	{attribute 'TcIecLibraryType'}
	{attribute 'external_name' := 'F_VN_TransformIntoDisplayableImage_GUID_02E0E048_CC89_5F60_6F70_D9022D4465A5'}
	(* Transform an image into a displayable image. The source image will be released and zeroed while existing destination images will be released and overwritten with the function result. The source image must not be used anywhere else and the transformation is very fast. If you want to use ipSrcImage after this function call, use F_VN_CopyIntoDisplayableImage instead. *)
	FUNCTION F_VN_TransformIntoDisplayableImage : HRESULT
	VAR_INPUT
		ipSrcImage	:	REFERENCE TO ITcVnImage;	(* Source image *)
		ipDestImage	:	REFERENCE TO ITcVnDisplayableImage;	(* Returns the displayable image *)
		hrPrev	:	HRESULT;	(* HRESULT indicating the result of previous operations (If SUCCEEDED(hrPrev) equals false, no operation is executed.) *)
	END_VAR

END_FUNCTION

// Functions/Basic Image Operations/F_VN_CreateAssociatedImage

	{attribute 'TcIecLibraryType'}
	{attribute 'external_name' := 'F_VN_CreateAssociatedImage_GUID_40D3B2A0_2CE9_5E22_5A39_BDDFD776A88E'}
	(* Creates a new image that shares its data with the source image. E.g. useful to work on different (disjoint) ROIs in parallel. *)
	FUNCTION F_VN_CreateAssociatedImage : HRESULT
	VAR_INPUT
		ipSrcImage	:	ITcVnImage;	(* Source image *)
		ipDestImage	:	REFERENCE TO ITcVnImage;	(* Returns the created image (Non-zero interface pointers are reused.) *)
		hrPrev	:	HRESULT;	(* HRESULT indicating the result of previous operations (If SUCCEEDED(hrPrev) equals false, no operation is executed.) *)
	END_VAR

END_FUNCTION

// Functions/Basic Image Operations/F_VN_CreateEmptyImage

	{attribute 'TcIecLibraryType'}
	{attribute 'external_name' := 'F_VN_CreateEmptyImage_GUID_87DE2717_AD60_5E53_651E_5AB98332C7FD'}
	(* Creates an empty image without allocating any data buffer. The initial reference count is set to one if a new image interface is created and kept, otherwise. *)
	FUNCTION F_VN_CreateEmptyImage : HRESULT
	VAR_INPUT
		ipImage	:	REFERENCE TO ITcVnImage;	(* Returns the created image *)
		hrPrev	:	HRESULT;	(* HRESULT indicating the result of previous operations (If SUCCEEDED(hrPrev) equals false, no operation is executed.) *)
	END_VAR

END_FUNCTION

// Functions/Basic Image Operations/F_VN_CreateImage

	{attribute 'TcIecLibraryType'}
	{attribute 'external_name' := 'F_VN_CreateImage_GUID_8D7420DD_6F30_56B3_5361_D2A5604ACF86'}
	(* Creates an image and allocate an appropriate data buffer. The initial reference count is set to one if a new image interface is created and kept, otherwise. *)
	FUNCTION F_VN_CreateImage : HRESULT
	VAR_INPUT
		ipImage	:	REFERENCE TO ITcVnImage;	(* Returns the created image (Non-zero interface pointers are reused.) *)
		nWidth	:	UDINT;	(* Image width *)
		nHeight	:	UDINT;	(* Image height *)
		ePixelType	:	ETcVnElementType;	(* Pixel type *)
		nChannelNum	:	UDINT;	(* Number of channels (1 to 255) *)
		hrPrev	:	HRESULT;	(* HRESULT indicating the result of previous operations (If SUCCEEDED(hrPrev) equals false, no operation is executed.) *)
	END_VAR

END_FUNCTION

// Functions/Basic Image Operations/F_VN_CreateImageAndSetPixels

	{attribute 'TcIecLibraryType'}
	{attribute 'external_name' := 'F_VN_CreateImageAndSetPixels_GUID_A8920FF8_8F96_5FBC_52F3_92CD14F74A4F'}
	(* Creates an image, allocates an appropriate data buffer and sets all pixels to the specified value. The initial reference count is set to one if a new image interface is created and kept, otherwise. *)
	FUNCTION F_VN_CreateImageAndSetPixels : HRESULT
	VAR_INPUT
		ipImage	:	REFERENCE TO ITcVnImage;	(* Returns the created image (Non-zero interface pointers are reused.) *)
		nWidth	:	UDINT;	(* Image width *)
		nHeight	:	UDINT;	(* Image height *)
		ePixelType	:	ETcVnElementType;	(* Pixel type *)
		nChannelNum	:	UDINT;	(* Number of channels (1 to 4) *)
		aValue	:	REFERENCE TO TcVnVector4_LREAL;	(* Pixel value *)
		hrPrev	:	HRESULT;	(* HRESULT indicating the result of previous operations (If SUCCEEDED(hrPrev) equals false, no operation is executed.) *)
	END_VAR

END_FUNCTION

// Functions/Basic Image Operations/F_VN_CreateImageFromArray

	{attribute 'TcIecLibraryType'}
	{attribute 'external_name' := 'F_VN_CreateImageFromArray_GUID_61CDDD3E_1106_53D6_5356_1EDFAEADE3E0'}
	(* Creates an image and initialize it with the provided data. The initial reference count is set to one if a new image interface is created and kept, otherwise. *)
	FUNCTION F_VN_CreateImageFromArray : HRESULT
	VAR_INPUT
		pData	:	PVOID;	(* Pointer to the 1D data array. Make sure that the array contains at least nWidth * nHeight * nChannelNum elements and that the array element type matches ePixelType. *)
		ipImage	:	REFERENCE TO ITcVnImage;	(* Returns the created image (Non-zero interface pointers are reused.) *)
		nWidth	:	UDINT;	(* Image width *)
		nHeight	:	UDINT;	(* Image height *)
		ePixelType	:	ETcVnElementType;	(* Pixel type *)
		nChannelNum	:	UDINT;	(* Number of channels (1 to 255) *)
		hrPrev	:	HRESULT;	(* HRESULT indicating the result of previous operations (If SUCCEEDED(hrPrev) equals false, no operation is executed.) *)
	END_VAR

END_FUNCTION

// Functions/Basic Image Operations/F_VN_ExportImage

	{attribute 'TcIecLibraryType'}
	{attribute 'external_name' := 'F_VN_ExportImage_GUID_12937EAB_04EC_5AB4_58D9_551F14B67CB3'}
	(* Exports the image data into a given buffer (e.g. an array). F_VN_ExportImageSize should be called before to get the required buffer size. *)
	FUNCTION F_VN_ExportImage : HRESULT
	VAR_INPUT
		ipImage	:	ITcVnImage;	(* Image *)
		pBuffer	:	PVOID;	(* Pointer to a buffer to store the image data (Make sure to allocate enough memory! The required size in bytes can be determined using the function F_VN_ExportImageSize) *)
		nBufferSize	:	ULINT;	(* Size of the buffer memory in bytes *)
		hrPrev	:	HRESULT;	(* HRESULT indicating the result of previous operations (If SUCCEEDED(hrPrev) equals false, no operation is executed.) *)
	END_VAR

END_FUNCTION

// Functions/Basic Image Operations/F_VN_ExportImageSize

	{attribute 'TcIecLibraryType'}
	{attribute 'external_name' := 'F_VN_ExportImageSize_GUID_992C005D_F63B_55F7_7FBB_93717F8A23F0'}
	(* Get the required buffer size (in bytes) to store the image data. *)
	FUNCTION F_VN_ExportImageSize : HRESULT
	VAR_INPUT
		ipImage	:	ITcVnImage;	(* Image *)
		nBufferSize	:	REFERENCE TO ULINT;	(* Returns the required buffer size in bytes *)
		hrPrev	:	HRESULT;	(* HRESULT indicating the result of previous operations (If SUCCEEDED(hrPrev) equals false, no operation is executed.) *)
	END_VAR

END_FUNCTION

// Functions/Basic Image Operations/F_VN_ExportImageAsBmp

	{attribute 'TcIecLibraryType'}
	{attribute 'external_name' := 'F_VN_ExportImageAsBmp_GUID_4BCA8984_D078_540E_761E_EBF20019EFCB'}
	(* Exports the image as bitmap into a given buffer (e.g. an array). F_VN_ExportImageAsBmpSize should be called before to get the required buffer size. *)
	FUNCTION F_VN_ExportImageAsBmp : HRESULT
	VAR_INPUT
		ipImage	:	ITcVnImage;	(* Image *)
		pBuffer	:	PVOID;	(* Pointer to a buffer to store the bitmap image (Make sure to allocate enough memory! The required size in bytes can be determined using the function F_VN_ExportImageAsBmpSize) *)
		nBufferSize	:	ULINT;	(* Size of the buffer memory in bytes *)
		hrPrev	:	HRESULT;	(* HRESULT indicating the result of previous operations (If SUCCEEDED(hrPrev) equals false, no operation is executed.) *)
	END_VAR

END_FUNCTION

// Functions/Basic Image Operations/F_VN_ExportImageAsBmpSize

	{attribute 'TcIecLibraryType'}
	{attribute 'external_name' := 'F_VN_ExportImageAsBmpSize_GUID_0FD9F0BD_DE92_5963_6C27_50E4417ED287'}
	(* Get the required buffer size (in bytes) to store the image as bitmap. *)
	FUNCTION F_VN_ExportImageAsBmpSize : HRESULT
	VAR_INPUT
		ipImage	:	ITcVnImage;	(* Image *)
		nBufferSize	:	REFERENCE TO ULINT;	(* Returns the required buffer size in bytes *)
		hrPrev	:	HRESULT;	(* HRESULT indicating the result of previous operations (If SUCCEEDED(hrPrev) equals false, no operation is executed.) *)
	END_VAR

END_FUNCTION

// Functions/Basic Image Operations/F_VN_ExportImageAsBmpExp

	{attribute 'TcIecLibraryType'}
	{attribute 'external_name' := 'F_VN_ExportImageAsBmpExp_GUID_47731DB6_D34C_5D53_45C4_8849F5EA485D'}
	(* Exports the image as bitmap into a given buffer (e.g. an array). F_VN_ExportImageAsBmpSizeExp should be called before to get the required buffer size. (expert function) *)
	FUNCTION F_VN_ExportImageAsBmpExp : HRESULT
	VAR_INPUT
		ipImage	:	ITcVnImage;	(* Image *)
		pBuffer	:	PVOID;	(* Pointer to a buffer to store the bitmap image (Make sure to allocate enough memory! The required size in bytes can be determined using the function F_VN_ExportImageAsBmpSizeExp) *)
		nBufferSize	:	ULINT;	(* Size of the buffer memory in bytes *)
		nWidth	:	UDINT;	(* Desired width (or 0 to keep the original width) *)
		nHeight	:	UDINT;	(* Desired height (or 0 to keep the original height) *)
		hrPrev	:	HRESULT;	(* HRESULT indicating the result of previous operations (If SUCCEEDED(hrPrev) equals false, no operation is executed.) *)
	END_VAR

END_FUNCTION

// Functions/Basic Image Operations/F_VN_ExportImageAsBmpSizeExp

	{attribute 'TcIecLibraryType'}
	{attribute 'external_name' := 'F_VN_ExportImageAsBmpSizeExp_GUID_152A8073_1085_5FC6_79DE_8B29B49970A3'}
	(* Get the required buffer size (in bytes) to store the image as bitmap. (expert function) *)
	FUNCTION F_VN_ExportImageAsBmpSizeExp : HRESULT
	VAR_INPUT
		ipImage	:	ITcVnImage;	(* Image *)
		nBufferSize	:	REFERENCE TO ULINT;	(* Returns the required buffer size in bytes *)
		nWidth	:	UDINT;	(* Desired width (or 0 to keep the original width) *)
		nHeight	:	UDINT;	(* Desired height (or 0 to keep the original height) *)
		hrPrev	:	HRESULT;	(* HRESULT indicating the result of previous operations (If SUCCEEDED(hrPrev) equals false, no operation is executed.) *)
	END_VAR

END_FUNCTION

// Functions/Basic Image Operations/F_VN_FuseImages

	{attribute 'TcIecLibraryType'}
	{attribute 'external_name' := 'F_VN_FuseImages_GUID_44F73693_9DB3_5AEB_675B_C4C1A72A31C1'}
	(* Fuse 2 images vertically (intended for line scan cameras). *)
	FUNCTION F_VN_FuseImages : HRESULT
	VAR_INPUT
		ipSrcImage1	:	ITcVnImage;	(* Source image 1 *)
		ipSrcImage2	:	ITcVnImage;	(* Source image 2 *)
		ipDestImage	:	REFERENCE TO ITcVnImage;	(* Destination image *)
		nFirstLine	:	UDINT;	(* Line index in ipSrcImage1, which is the first line in ipDestImage *)
		nNumLines	:	UDINT;	(* The number of lines that should be copied to ipDestImage, starting with nFirstLine in ipSrcImage1. Once the last line of ipSrcImage1 was copied, the remaining lines are copied from ipSrcImage2, starting at line index 0. *)
		hrPrev	:	HRESULT;	(* HRESULT indicating the result of previous operations (If SUCCEEDED(hrPrev) equals false, no operation is executed.) *)
	END_VAR

END_FUNCTION

// Functions/Basic Image Operations/F_VN_FuseImagesArray

	{attribute 'TcIecLibraryType'}
	{attribute 'external_name' := 'F_VN_FuseImagesArray_GUID_70FE5178_8522_5DE6_63B0_CBF59E4BE48B'}
	(* Fuse up to 10 images vertically (intended for line scan cameras). *)
	FUNCTION F_VN_FuseImagesArray : HRESULT
	VAR_INPUT
		aSrcImageArray	:	REFERENCE TO TcVnArray10_ITcVnImage;	(* Ten-element source image array (not all elements need to be filled, nValidImages specifies the actual amount of images) *)
		nValidImages	:	UDINT;	(* Number of valid images in aSrcImageArray *)
		ipDestImage	:	REFERENCE TO ITcVnImage;	(* Destination image *)
		nFirstLine	:	UDINT;	(* Line index in ipSrcImage1, which is the first line in ipDestImage *)
		nNumLines	:	UDINT;	(* The number of lines that should be copied to ipDestImage, starting with nFirstLine in aSrcImageArray[0]. Once the last line of aSrcImageArray[0] was copied, the remaining lines are copied from aSrcImageArray[1] (starting at line index 0) and so on. *)
		hrPrev	:	HRESULT;	(* HRESULT indicating the result of previous operations (If SUCCEEDED(hrPrev) equals false, no operation is executed.) *)
	END_VAR

END_FUNCTION

// Functions/Basic Image Operations/F_VN_GetImageChannel

	{attribute 'TcIecLibraryType'}
	{attribute 'external_name' := 'F_VN_GetImageChannel_GUID_15192384_BD29_5960_5E27_71E33EA35C78'}
	(* Return the specified source image channel as a single-channel image. *)
	FUNCTION F_VN_GetImageChannel : HRESULT
	VAR_INPUT
		ipSrcImage	:	ITcVnImage;	(* Source image *)
		ipDestImage	:	REFERENCE TO ITcVnImage;	(* Destination image (An appropriate image will be created if required.) *)
		nChannelIndex	:	UINT;	(* Index of the requested source image channel *)
		hrPrev	:	HRESULT;	(* HRESULT indicating the result of previous operations (If SUCCEEDED(hrPrev) equals false, no operation is executed.) *)
	END_VAR

END_FUNCTION

// Functions/Basic Image Operations/F_VN_GetImageHeight

	{attribute 'TcIecLibraryType'}
	{attribute 'external_name' := 'F_VN_GetImageHeight_GUID_65DFE3C5_BA03_5A08_5064_B1CFB2712520'}
	(* Return the height of an image. (Alternatively use interface method .GetHeight.) *)
	FUNCTION F_VN_GetImageHeight : HRESULT
	VAR_INPUT
		ipImage	:	ITcVnImage;	(* Image *)
		nHeight	:	REFERENCE TO UDINT;	(* Return the height of ipImage *)
		hrPrev	:	HRESULT;	(* HRESULT indicating the result of previous operations (If SUCCEEDED(hrPrev) equals false, no operation is executed.) *)
	END_VAR

END_FUNCTION

// Functions/Basic Image Operations/F_VN_GetImageInfo

	{attribute 'TcIecLibraryType'}
	{attribute 'external_name' := 'F_VN_GetImageInfo_GUID_24926DD3_FE67_5D84_418A_8B86040FF853'}
	(* Gets a struct containing all common meta infos of the image. (Alternatively use interface method .GetImageInfo.) *)
	FUNCTION F_VN_GetImageInfo : HRESULT
	VAR_INPUT
		ipImage	:	ITcVnImage;	(* Image *)
		stImageInfo	:	REFERENCE TO TcVnImageInfo;	(* Returns a struct describing the image *)
		hrPrev	:	HRESULT;	(* HRESULT indicating the result of previous operations (If SUCCEEDED(hrPrev) equals false, no operation is executed.) *)
	END_VAR

END_FUNCTION

// Functions/Basic Image Operations/F_VN_GetImageWidth

	{attribute 'TcIecLibraryType'}
	{attribute 'external_name' := 'F_VN_GetImageWidth_GUID_5D3D1FA2_8F31_560E_4CB0_2AA032E1BECA'}
	(* Return the width of an image. (Alternatively use interface method .GetWidth.) *)
	FUNCTION F_VN_GetImageWidth : HRESULT
	VAR_INPUT
		ipImage	:	ITcVnImage;	(* Image *)
		nWidth	:	REFERENCE TO UDINT;	(* Return the width of ipImage *)
		hrPrev	:	HRESULT;	(* HRESULT indicating the result of previous operations (If SUCCEEDED(hrPrev) equals false, no operation is executed.) *)
	END_VAR

END_FUNCTION

// Functions/Basic Image Operations/F_VN_GetPixel

	{attribute 'TcIecLibraryType'}
	{attribute 'external_name' := 'F_VN_GetPixel_GUID_5FD4139A_8160_5C6E_5BE9_914D15E9AEEF'}
	(* Gets a specific pixel. *)
	FUNCTION F_VN_GetPixel : HRESULT
	VAR_INPUT
		ipSrcImage	:	ITcVnImage;	(* Source image *)
		aValue	:	REFERENCE TO TcVnVector4_LREAL;	(* Returns the pixel value (Unused channels are set to 0.) *)
		nX	:	UDINT;	(* x coordinate of the pixel *)
		nY	:	UDINT;	(* y coordinate of the pixel *)
		hrPrev	:	HRESULT;	(* HRESULT indicating the result of previous operations (If SUCCEEDED(hrPrev) equals false, no operation is executed.) *)
	END_VAR

END_FUNCTION

// Functions/Basic Image Operations/F_VN_GetPixelFormat

	{attribute 'TcIecLibraryType'}
	{attribute 'external_name' := 'F_VN_GetPixelFormat_GUID_D4DC166C_AD15_5B86_63E1_7B44C8A4886C'}
	(* Gets the pixel format of an image. (Alternatively use interface method .GetPixelFormat.) *)
	FUNCTION F_VN_GetPixelFormat : HRESULT
	VAR_INPUT
		ipImage	:	ITcVnImage;	(* Image *)
		stPixelFormat	:	REFERENCE TO TcVnPixelFormat;	(* Returns a struct describing the pixel format *)
		hrPrev	:	HRESULT;	(* HRESULT indicating the result of previous operations (If SUCCEEDED(hrPrev) equals false, no operation is executed.) *)
	END_VAR

END_FUNCTION

// Functions/Basic Image Operations/F_VN_GetRoi

	{attribute 'TcIecLibraryType'}
	{attribute 'external_name' := 'F_VN_GetRoi_GUID_177883C9_0780_5F81_589B_F315CCBE5526'}
	(* Gets the coordinates of the region of interest (ROI) within the image. *)
	FUNCTION F_VN_GetRoi : HRESULT
	VAR_INPUT
		ipSrcImage	:	ITcVnImage;	(* Source image *)
		stRoi	:	REFERENCE TO TcVnRectangle_UDINT;	(* Returns the coordinates of the region of interest *)
		hrPrev	:	HRESULT;	(* HRESULT indicating the result of previous operations (If SUCCEEDED(hrPrev) equals false, no operation is executed.) *)
	END_VAR

END_FUNCTION

// Functions/Basic Image Operations/F_VN_MixImageChannels

	{attribute 'TcIecLibraryType'}
	{attribute 'external_name' := 'F_VN_MixImageChannels_GUID_11F8244D_387D_5591_7A84_7EC6ED704714'}
	(* Mix image channels by copying the specified channels of the source image into the specified channels of the destination image. *)
	FUNCTION F_VN_MixImageChannels : HRESULT
	VAR_INPUT
		ipSrcImage	:	ITcVnImage;	(* Source image *)
		ipDestImage	:	REFERENCE TO ITcVnImage;	(* Destination image (An appropriate image will be created if required.) *)
		ipIndicesFromTo	:	ITcVnContainer;	(* Index pairs (ContainerType_Vector_TcVnVector2_DINT), specifying which source channel (TcVnVector2_DINT [0]) should be copied to which destination channel (TcVnVector2_DINT [1]). *)
		hrPrev	:	HRESULT;	(* HRESULT indicating the result of previous operations (If SUCCEEDED(hrPrev) equals false, no operation is executed.) *)
	END_VAR

END_FUNCTION

// Functions/Basic Image Operations/F_VN_ResetRoi

	{attribute 'TcIecLibraryType'}
	{attribute 'external_name' := 'F_VN_ResetRoi_GUID_C7E8B0BE_2056_5152_456B_BF1D4597B825'}
	(* Reset the region of interest (ROI) of an image. (After this operation, the ROI is set to the entire image.) *)
	FUNCTION F_VN_ResetRoi : HRESULT
	VAR_INPUT
		ipImage	:	ITcVnImage;	(* Image *)
		hrPrev	:	HRESULT;	(* HRESULT indicating the result of previous operations (If SUCCEEDED(hrPrev) equals false, no operation is executed.) *)
	END_VAR

END_FUNCTION

// Functions/Basic Image Operations/F_VN_SetImageChannel

	{attribute 'TcIecLibraryType'}
	{attribute 'external_name' := 'F_VN_SetImageChannel_GUID_E1A99947_7DDD_5872_6D1A_8654E9EE7820'}
	(* Sets the specified destination image channel to the values of the specified source image channel. *)
	FUNCTION F_VN_SetImageChannel : HRESULT
	VAR_INPUT
		ipSrcImage	:	ITcVnImage;	(* Source image *)
		ipDestImage	:	REFERENCE TO ITcVnImage;	(* Destination image (An appropriate image will be created if required.) *)
		nSrcChannelIndex	:	UINT;	(* Index of the source image channel *)
		nDestChannelIndex	:	UINT;	(* Index of the destination image channel, which will be replaced by the specified source image channel *)
		hrPrev	:	HRESULT;	(* HRESULT indicating the result of previous operations (If SUCCEEDED(hrPrev) equals false, no operation is executed.) *)
	END_VAR

END_FUNCTION

// Functions/Basic Image Operations/F_VN_SetPixel

	{attribute 'TcIecLibraryType'}
	{attribute 'external_name' := 'F_VN_SetPixel_GUID_60FCB15E_2791_5C28_4A1C_2D15B1A56113'}
	(* Sets a specific pixel. *)
	FUNCTION F_VN_SetPixel : HRESULT
	VAR_INPUT
		ipSrcImage	:	ITcVnImage;	(* Source image *)
		aValue	:	REFERENCE TO TcVnVector4_LREAL;	(* The pixel value to set (additional channels are ignored.) *)
		nX	:	UDINT;	(* x coordinate of the pixel *)
		nY	:	UDINT;	(* y coordinate of the pixel *)
		hrPrev	:	HRESULT;	(* HRESULT indicating the result of previous operations (If SUCCEEDED(hrPrev) equals false, no operation is executed.) *)
	END_VAR

END_FUNCTION

// Functions/Basic Image Operations/F_VN_SetPixels

	{attribute 'TcIecLibraryType'}
	{attribute 'external_name' := 'F_VN_SetPixels_GUID_115B93BA_4340_52EC_4CF7_374B90A64A2C'}
	(* Sets all pixels of an image to a given value. *)
	FUNCTION F_VN_SetPixels : HRESULT
	VAR_INPUT
		ipDestImage	:	ITcVnImage;	(* Destination image *)
		aValue	:	REFERENCE TO TcVnVector4_LREAL;	(* Pixel value *)
		hrPrev	:	HRESULT;	(* HRESULT indicating the result of previous operations (If SUCCEEDED(hrPrev) equals false, no operation is executed.) *)
	END_VAR

END_FUNCTION

// Functions/Basic Image Operations/F_VN_SetPixelsExp

	{attribute 'TcIecLibraryType'}
	{attribute 'external_name' := 'F_VN_SetPixelsExp_GUID_AE738DF5_656D_5E40_586E_C2535624EFB6'}
	(* Sets all pixels of an image to a given value. (expert function) *)
	FUNCTION F_VN_SetPixelsExp : HRESULT
	VAR_INPUT
		ipDestImage	:	ITcVnImage;	(* Destination image *)
		aValue	:	REFERENCE TO TcVnVector4_LREAL;	(* Pixel value *)
		ipMask	:	ITcVnImage;	(* Mask image *)
		hrPrev	:	HRESULT;	(* HRESULT indicating the result of previous operations (If SUCCEEDED(hrPrev) equals false, no operation is executed.) *)
	END_VAR

END_FUNCTION

// Functions/Basic Image Operations/F_VN_SetRoi

	{attribute 'TcIecLibraryType'}
	{attribute 'external_name' := 'F_VN_SetRoi_GUID_80E727B0_F5BF_5833_50F3_048E61BC1216'}
	(* Sets a region of interest (ROI) within an image. *)
	FUNCTION F_VN_SetRoi : HRESULT
	VAR_INPUT
		nX	:	UDINT;	(* Left boundary (inclusive 0-based index) *)
		nY	:	UDINT;	(* Upper boundary (inclusive 0-based index) *)
		nWidth	:	UDINT;	(* ROI width *)
		nHeight	:	UDINT;	(* ROI height *)
		ipDestImage	:	ITcVnImage;	(* Destination image *)
		hrPrev	:	HRESULT;	(* HRESULT indicating the result of previous operations (If SUCCEEDED(hrPrev) equals false, no operation is executed.) *)
	END_VAR

END_FUNCTION

// Functions/Basic Image Operations/F_VN_SetRoi_TcVnRectangle_UDINT

	{attribute 'TcIecLibraryType'}
	{attribute 'external_name' := 'F_VN_SetRoi_TcVnRectangle_UDINT_GUID_8B9629C2_0057_5448_4E0E_2D25120D6927'}
	(* Sets a region of interest (ROI) within an image. *)
	FUNCTION F_VN_SetRoi_TcVnRectangle_UDINT : HRESULT
	VAR_INPUT
		stRoi	:	REFERENCE TO TcVnRectangle_UDINT;	(* Region of interest *)
		ipDestImage	:	ITcVnImage;	(* Destination image *)
		hrPrev	:	HRESULT;	(* HRESULT indicating the result of previous operations (If SUCCEEDED(hrPrev) equals false, no operation is executed.) *)
	END_VAR

END_FUNCTION

// Functions/Basic Image Operations/F_VN_SplitImageChannels

	{attribute 'TcIecLibraryType'}
	{attribute 'external_name' := 'F_VN_SplitImageChannels_GUID_42E612CB_D027_57DD_5C9B_A3E0227F93DF'}
	(* Split a multi-channel image into multiple single channel images (1 for each source image channel). *)
	FUNCTION F_VN_SplitImageChannels : HRESULT
	VAR_INPUT
		ipSrcImage	:	ITcVnImage;	(* Source image with multiple channels *)
		pDestImages	:	PVOID;	(* Pointer to an array of single-channel destination images (appropriate destination images will be created if required.) *)
		nArraySize	:	UINT;	(* pDestImages array size (at least the number or source image channels required) *)
		hrPrev	:	HRESULT;	(* HRESULT indicating the result of previous operations (If SUCCEEDED(hrPrev) equals false, no operation is executed.) *)
	END_VAR
	VAR_OUTPUT
		nImageChannels	:	UINT;	(* Actual source image channels *)
	END_VAR

END_FUNCTION

// Functions/Basic Image Operations/F_VN_TransformIntoDisplayableImageExp

	{attribute 'TcIecLibraryType'}
	{attribute 'external_name' := 'F_VN_TransformIntoDisplayableImageExp_GUID_FDC2D0E3_3C06_5CB4_56AF_120A5601EFA8'}
	(* Transform an image into a displayable image. The source image will be released and zeroed while existing destination images will be released and overwritten with the function result. If bAllowDeepCopy equals false, the source image must not be used anywhere else and the transformation is always very fast. Otherwise, if bAllowDeepCopy equals true, a deep copy of the source image might be created if required, which will result in a longer execution time. If you want to use ipSrcImage after this function call, use F_VN_CopyIntoDisplayableImage instead. (expert function) *)
	FUNCTION F_VN_TransformIntoDisplayableImageExp : HRESULT
	VAR_INPUT
		ipSrcImage	:	REFERENCE TO ITcVnImage;	(* Source image *)
		ipDestImage	:	REFERENCE TO ITcVnDisplayableImage;	(* Returns the displayable image *)
		bAllowDeepCopy	:	BOOL;	(* Allow deep image copies, if required *)
		hrPrev	:	HRESULT;	(* HRESULT indicating the result of previous operations (If SUCCEEDED(hrPrev) equals false, no operation is executed.) *)
	END_VAR

END_FUNCTION

// Functions/Container Statistics/F_VN_ContainerAverage

	{attribute 'TcIecLibraryType'}
	{attribute 'external_name' := 'F_VN_ContainerAverage_GUID_41307245_B8D5_5CBF_7DE8_4781D77E9B35'}
	(* Calculate the average of elements in a container. *)
	FUNCTION F_VN_ContainerAverage : HRESULT
	VAR_INPUT
		ipSrcContainer	:	ITcVnContainer;	(* Source container (Arithmetic, point and vector element types are supported. For points and vectors, the euclidean norm is used.) *)
		fAverage	:	REFERENCE TO LREAL;	(* Returns the calculated average value *)
		hrPrev	:	HRESULT;	(* HRESULT indicating the result of previous operations (If SUCCEEDED(hrPrev) equals false, no operation is executed.) *)
	END_VAR

END_FUNCTION

// Functions/Container Statistics/F_VN_ContainerAverageElementwise2

	{attribute 'TcIecLibraryType'}
	{attribute 'external_name' := 'F_VN_ContainerAverageElementwise2_GUID_4E2EC21A_684C_5E48_7452_C3B7DF053377'}
	(* Calculate the elementwise average of 2D elements in a container. *)
	FUNCTION F_VN_ContainerAverageElementwise2 : HRESULT
	VAR_INPUT
		ipSrcContainer	:	ITcVnContainer;	(* Source container with 2D points or vectors *)
		aAverage	:	REFERENCE TO TcVnVector2_LREAL;	(* Returns the calculated average values *)
		hrPrev	:	HRESULT;	(* HRESULT indicating the result of previous operations (If SUCCEEDED(hrPrev) equals false, no operation is executed.) *)
	END_VAR

END_FUNCTION

// Functions/Container Statistics/F_VN_ContainerAverageElementwise3

	{attribute 'TcIecLibraryType'}
	{attribute 'external_name' := 'F_VN_ContainerAverageElementwise3_GUID_AB461934_6535_5419_517B_924C4B9DB715'}
	(* Calculate the elementwise average of 3D elements in a container. *)
	FUNCTION F_VN_ContainerAverageElementwise3 : HRESULT
	VAR_INPUT
		ipSrcContainer	:	ITcVnContainer;	(* Source container with 3D points or vectors *)
		aAverage	:	REFERENCE TO TcVnVector3_LREAL;	(* Returns the calculated average values *)
		hrPrev	:	HRESULT;	(* HRESULT indicating the result of previous operations (If SUCCEEDED(hrPrev) equals false, no operation is executed.) *)
	END_VAR

END_FUNCTION

// Functions/Container Statistics/F_VN_ContainerAverageElementwise4

	{attribute 'TcIecLibraryType'}
	{attribute 'external_name' := 'F_VN_ContainerAverageElementwise4_GUID_3514B60E_D784_5DED_78E6_3BEDF9ABC677'}
	(* Calculate the elementwise average of 4D elements in a container. *)
	FUNCTION F_VN_ContainerAverageElementwise4 : HRESULT
	VAR_INPUT
		ipSrcContainer	:	ITcVnContainer;	(* Source container with 4D vectors *)
		aAverage	:	REFERENCE TO TcVnVector4_LREAL;	(* Returns the calculated average values *)
		hrPrev	:	HRESULT;	(* HRESULT indicating the result of previous operations (If SUCCEEDED(hrPrev) equals false, no operation is executed.) *)
	END_VAR

END_FUNCTION

// Functions/Container Statistics/F_VN_ContainerAverageVariance

	{attribute 'TcIecLibraryType'}
	{attribute 'external_name' := 'F_VN_ContainerAverageVariance_GUID_13D51E0F_284F_50C1_731C_E633EA49E595'}
	(* Calculate the average and variance of elements in a container. *)
	FUNCTION F_VN_ContainerAverageVariance : HRESULT
	VAR_INPUT
		ipSrcContainer	:	ITcVnContainer;	(* Source container (Arithmetic, point and vector element types are supported. For points and vectors, the euclidean norm is used.) *)
		fAverage	:	REFERENCE TO LREAL;	(* Returns the calculated average value *)
		fVariance	:	REFERENCE TO LREAL;	(* Returns the calculated variance value *)
		hrPrev	:	HRESULT;	(* HRESULT indicating the result of previous operations (If SUCCEEDED(hrPrev) equals false, no operation is executed.) *)
	END_VAR

END_FUNCTION

// Functions/Container Statistics/F_VN_ContainerAverageVarianceElementwise2

	{attribute 'TcIecLibraryType'}
	{attribute 'external_name' := 'F_VN_ContainerAverageVarianceElementwise2_GUID_76609C44_F3A1_5B34_7E40_9B6235BAEC4C'}
	(* Calculate the elementwise average and variance of 2D elements in a container. *)
	FUNCTION F_VN_ContainerAverageVarianceElementwise2 : HRESULT
	VAR_INPUT
		ipSrcContainer	:	ITcVnContainer;	(* Source container with 2D points or vectors *)
		aAverage	:	REFERENCE TO TcVnVector2_LREAL;	(* Returns the calculated average values *)
		aVariance	:	REFERENCE TO TcVnVector2_LREAL;	(* Returns the calculated variance values *)
		hrPrev	:	HRESULT;	(* HRESULT indicating the result of previous operations (If SUCCEEDED(hrPrev) equals false, no operation is executed.) *)
	END_VAR

END_FUNCTION

// Functions/Container Statistics/F_VN_ContainerAverageVarianceElementwise3

	{attribute 'TcIecLibraryType'}
	{attribute 'external_name' := 'F_VN_ContainerAverageVarianceElementwise3_GUID_113B12EB_43D5_53D9_6BDC_56E4656A0370'}
	(* Calculate the elementwise average and variance of 3D elements in a container. *)
	FUNCTION F_VN_ContainerAverageVarianceElementwise3 : HRESULT
	VAR_INPUT
		ipSrcContainer	:	ITcVnContainer;	(* Source container with 3D points or vectors *)
		aAverage	:	REFERENCE TO TcVnVector3_LREAL;	(* Returns the calculated average values *)
		aVariance	:	REFERENCE TO TcVnVector3_LREAL;	(* Returns the calculated variance values *)
		hrPrev	:	HRESULT;	(* HRESULT indicating the result of previous operations (If SUCCEEDED(hrPrev) equals false, no operation is executed.) *)
	END_VAR

END_FUNCTION

// Functions/Container Statistics/F_VN_ContainerAverageVarianceElementwise4

	{attribute 'TcIecLibraryType'}
	{attribute 'external_name' := 'F_VN_ContainerAverageVarianceElementwise4_GUID_E8A65177_F1B0_5D00_4264_079550CA1D3C'}
	(* Calculate the elementwise average and variance of 4D elements in a container. *)
	FUNCTION F_VN_ContainerAverageVarianceElementwise4 : HRESULT
	VAR_INPUT
		ipSrcContainer	:	ITcVnContainer;	(* Source container with 4D vectors *)
		aAverage	:	REFERENCE TO TcVnVector4_LREAL;	(* Returns the calculated average values *)
		aVariance	:	REFERENCE TO TcVnVector4_LREAL;	(* Returns the calculated variance values *)
		hrPrev	:	HRESULT;	(* HRESULT indicating the result of previous operations (If SUCCEEDED(hrPrev) equals false, no operation is executed.) *)
	END_VAR

END_FUNCTION

// Functions/Container Statistics/F_VN_MaxElement

	{attribute 'TcIecLibraryType'}
	{attribute 'external_name' := 'F_VN_MaxElement_GUID_78EBF024_AA4F_5222_5208_3A9186A36222'}
	(* Gets the maximum element of a container. *)
	FUNCTION F_VN_MaxElement : HRESULT
	VAR_INPUT
		ipSrcContainer	:	ITcVnContainer;	(* Source container (Arithmetic, point and vector element types are supported. For points and vectors, the euclidean norm is used.) *)
		ipDestIterator	:	REFERENCE TO ITcVnBidirectionalIterator;	(* Returns an iterator to the requested element *)
		nIndex	:	REFERENCE TO ULINT;	(* Returns the position of the requested element within the container *)
		hrPrev	:	HRESULT;	(* HRESULT indicating the result of previous operations (If SUCCEEDED(hrPrev) equals false, no operation is executed.) *)
	END_VAR

END_FUNCTION

// Functions/Container Statistics/F_VN_MedianElement

	{attribute 'TcIecLibraryType'}
	{attribute 'external_name' := 'F_VN_MedianElement_GUID_98FE4FA7_BE0E_5C67_4975_9A043C80412B'}
	(* Gets the median element of a container. *)
	FUNCTION F_VN_MedianElement : HRESULT
	VAR_INPUT
		ipSrcContainer	:	ITcVnContainer;	(* Source container (Arithmetic, point and vector element types are supported. For points and vectors, the euclidean norm is used.) *)
		ipDestIterator	:	REFERENCE TO ITcVnBidirectionalIterator;	(* Returns an iterator to the requested element *)
		nIndex	:	REFERENCE TO ULINT;	(* Returns the position of the requested element within the container *)
		hrPrev	:	HRESULT;	(* HRESULT indicating the result of previous operations (If SUCCEEDED(hrPrev) equals false, no operation is executed.) *)
	END_VAR

END_FUNCTION

// Functions/Container Statistics/F_VN_MinElement

	{attribute 'TcIecLibraryType'}
	{attribute 'external_name' := 'F_VN_MinElement_GUID_7EDBAD44_AE62_5012_763A_9695CCB1740C'}
	(* Gets the minimum element of a container. *)
	FUNCTION F_VN_MinElement : HRESULT
	VAR_INPUT
		ipSrcContainer	:	ITcVnContainer;	(* Source container (Arithmetic, point and vector element types are supported. For points and vectors, the euclidean norm is used.) *)
		ipDestIterator	:	REFERENCE TO ITcVnBidirectionalIterator;	(* Returns an iterator to the requested element *)
		nIndex	:	REFERENCE TO ULINT;	(* Returns the position of the requested element within the container *)
		hrPrev	:	HRESULT;	(* HRESULT indicating the result of previous operations (If SUCCEEDED(hrPrev) equals false, no operation is executed.) *)
	END_VAR

END_FUNCTION

// Functions/Fourier Analysis/F_VN_CreateBandpassButterworthFilter

	{attribute 'TcIecLibraryType'}
	{attribute 'external_name' := 'F_VN_CreateBandpassButterworthFilter_GUID_4FC9D2B4_135E_51B3_7419_B6FE646193A4'}
	(* Creates a bandpass Butterworth filter, which can be applied to a frequency domain image by element-wise multiplication. *)
	FUNCTION F_VN_CreateBandpassButterworthFilter : HRESULT
	VAR_INPUT
		ipFilter	:	REFERENCE TO ITcVnImage;	(* Returns the created filter (1 channel of type REAL or LREAL, depending on bDoublePrecision. Non-zero interface pointers are reused.). *)
		nWidth	:	UDINT;	(* Filter width (even, >= 2, must match the width of the image it is applied to) *)
		nHeight	:	UDINT;	(* Filter height (even, >= 2, must match the height of the image it is applied to) *)
		bDoublePrecision	:	BOOL;	(* If true, the filter is generated with double precision (LREAL) instead of single precision (REAL). *)
		bOriginAtCenter	:	BOOL;	(* If true, the filter origin is shifted to the image center. *)
		fCutoffDistance	:	LREAL;	(* The cutoff distance of the Butterworth filter (> 0). *)
		fBandWidth	:	LREAL;	(* The band width of the Butterworth filter (> 0). *)
		nOrder	:	UDINT;	(* The order of the Butterworth filter (> 0). *)
		fScale	:	LREAL;	(* The scale factor of the Butterworth filter denominator term (> 0, e.g. 0.414 or 1.0). *)
		hrPrev	:	HRESULT;	(* HRESULT indicating the result of previous operations (If SUCCEEDED(hrPrev) equals false, no operation is executed.) *)
	END_VAR

END_FUNCTION

// Functions/Fourier Analysis/F_VN_CreateBandpassGaussianFilter

	{attribute 'TcIecLibraryType'}
	{attribute 'external_name' := 'F_VN_CreateBandpassGaussianFilter_GUID_40864679_21AD_52CD_46CB_A097BA33545B'}
	(* Creates a bandpass Gaussian filter, which can be applied to a frequency domain image by element-wise multiplication. *)
	FUNCTION F_VN_CreateBandpassGaussianFilter : HRESULT
	VAR_INPUT
		ipFilter	:	REFERENCE TO ITcVnImage;	(* Returns the created filter (1 channel of type REAL or LREAL, depending on bDoublePrecision. Non-zero interface pointers are reused.). *)
		nWidth	:	UDINT;	(* Filter width (even, >= 2, must match the width of the image it is applied to) *)
		nHeight	:	UDINT;	(* Filter height (even, >= 2, must match the height of the image it is applied to) *)
		bDoublePrecision	:	BOOL;	(* If true, the filter is generated with double precision (LREAL) instead of single precision (REAL). *)
		bOriginAtCenter	:	BOOL;	(* If true, the filter origin is shifted to the image center. *)
		fCutoffDistance	:	LREAL;	(* The cutoff distance of the Gaussian filter (> 0). *)
		fBandWidth	:	LREAL;	(* The band width of the Gaussian filter (> 0). *)
		hrPrev	:	HRESULT;	(* HRESULT indicating the result of previous operations (If SUCCEEDED(hrPrev) equals false, no operation is executed.) *)
	END_VAR

END_FUNCTION

// Functions/Fourier Analysis/F_VN_CreateBandrejectButterworthFilter

	{attribute 'TcIecLibraryType'}
	{attribute 'external_name' := 'F_VN_CreateBandrejectButterworthFilter_GUID_A84545FC_B925_5054_58D1_2BF0DE2FA2E5'}
	(* Creates a bandreject Butterworth filter, which can be applied to a frequency domain image by element-wise multiplication. *)
	FUNCTION F_VN_CreateBandrejectButterworthFilter : HRESULT
	VAR_INPUT
		ipFilter	:	REFERENCE TO ITcVnImage;	(* Returns the created filter (1 channel of type REAL or LREAL, depending on bDoublePrecision. Non-zero interface pointers are reused.). *)
		nWidth	:	UDINT;	(* Filter width (even, >= 2, must match the width of the image it is applied to) *)
		nHeight	:	UDINT;	(* Filter height (even, >= 2, must match the height of the image it is applied to) *)
		bDoublePrecision	:	BOOL;	(* If true, the filter is generated with double precision (LREAL) instead of single precision (REAL). *)
		bOriginAtCenter	:	BOOL;	(* If true, the filter origin is shifted to the image center. *)
		fCutoffDistance	:	LREAL;	(* The cutoff distance of the Butterworth filter (> 0). *)
		fBandWidth	:	LREAL;	(* The band width of the Butterworth filter (> 0). *)
		nOrder	:	UDINT;	(* The order of the Butterworth filter (> 0). *)
		fScale	:	LREAL;	(* The scale factor of the Butterworth filter denominator term (> 0, e.g. 0.414 or 1.0). *)
		hrPrev	:	HRESULT;	(* HRESULT indicating the result of previous operations (If SUCCEEDED(hrPrev) equals false, no operation is executed.) *)
	END_VAR

END_FUNCTION

// Functions/Fourier Analysis/F_VN_CreateBandrejectGaussianFilter

	{attribute 'TcIecLibraryType'}
	{attribute 'external_name' := 'F_VN_CreateBandrejectGaussianFilter_GUID_C6BB47BB_4798_5264_48B3_6E757601C426'}
	(* Creates a bandreject Gaussian filter, which can be applied to a frequency domain image by element-wise multiplication. *)
	FUNCTION F_VN_CreateBandrejectGaussianFilter : HRESULT
	VAR_INPUT
		ipFilter	:	REFERENCE TO ITcVnImage;	(* Returns the created filter (1 channel of type REAL or LREAL, depending on bDoublePrecision. Non-zero interface pointers are reused.). *)
		nWidth	:	UDINT;	(* Filter width (even, >= 2, must match the width of the image it is applied to) *)
		nHeight	:	UDINT;	(* Filter height (even, >= 2, must match the height of the image it is applied to) *)
		bDoublePrecision	:	BOOL;	(* If true, the filter is generated with double precision (LREAL) instead of single precision (REAL). *)
		bOriginAtCenter	:	BOOL;	(* If true, the filter origin is shifted to the image center. *)
		fCutoffDistance	:	LREAL;	(* The cutoff distance of the Gaussian filter (> 0). *)
		fBandWidth	:	LREAL;	(* The band width of the Gaussian filter (> 0). *)
		hrPrev	:	HRESULT;	(* HRESULT indicating the result of previous operations (If SUCCEEDED(hrPrev) equals false, no operation is executed.) *)
	END_VAR

END_FUNCTION

// Functions/Fourier Analysis/F_VN_CreateHighpassButterworthFilter

	{attribute 'TcIecLibraryType'}
	{attribute 'external_name' := 'F_VN_CreateHighpassButterworthFilter_GUID_CD891381_4721_5C30_5F2F_C62B2AA2F74D'}
	(* Creates a highpass Butterworth filter, which can be applied to a frequency domain image by element-wise multiplication. *)
	FUNCTION F_VN_CreateHighpassButterworthFilter : HRESULT
	VAR_INPUT
		ipFilter	:	REFERENCE TO ITcVnImage;	(* Returns the created filter (1 channel of type REAL or LREAL, depending on bDoublePrecision. Non-zero interface pointers are reused.). *)
		nWidth	:	UDINT;	(* Filter width (even, >= 2, must match the width of the image it is applied to) *)
		nHeight	:	UDINT;	(* Filter height (even, >= 2, must match the height of the image it is applied to) *)
		bDoublePrecision	:	BOOL;	(* If true, the filter is generated with double precision (LREAL) instead of single precision (REAL). *)
		bOriginAtCenter	:	BOOL;	(* If true, the filter origin is shifted to the image center. *)
		fCutoffDistance	:	LREAL;	(* The cutoff distance of the Butterworth filter (> 0). *)
		nOrder	:	UDINT;	(* The order of the Butterworth filter (> 0). *)
		fScale	:	LREAL;	(* The scale factor of the Butterworth filter denominator term (> 0, e.g. 0.414 or 1.0). *)
		hrPrev	:	HRESULT;	(* HRESULT indicating the result of previous operations (If SUCCEEDED(hrPrev) equals false, no operation is executed.) *)
	END_VAR

END_FUNCTION

// Functions/Fourier Analysis/F_VN_CreateHighpassGaussianFilter

	{attribute 'TcIecLibraryType'}
	{attribute 'external_name' := 'F_VN_CreateHighpassGaussianFilter_GUID_7A0D8DA0_CD02_503D_7E7F_E212508066BC'}
	(* Creates a highpass Gaussian filter, which can be applied to a frequency domain image by element-wise multiplication. *)
	FUNCTION F_VN_CreateHighpassGaussianFilter : HRESULT
	VAR_INPUT
		ipFilter	:	REFERENCE TO ITcVnImage;	(* Returns the created filter (1 channel of type REAL or LREAL, depending on bDoublePrecision. Non-zero interface pointers are reused.). *)
		nWidth	:	UDINT;	(* Filter width (even, >= 2, must match the width of the image it is applied to) *)
		nHeight	:	UDINT;	(* Filter height (even, >= 2, must match the height of the image it is applied to) *)
		bDoublePrecision	:	BOOL;	(* If true, the filter is generated with double precision (LREAL) instead of single precision (REAL). *)
		bOriginAtCenter	:	BOOL;	(* If true, the filter origin is shifted to the image center. *)
		fCutoffDistance	:	LREAL;	(* The cutoff distance of the Gaussian filter (> 0). *)
		hrPrev	:	HRESULT;	(* HRESULT indicating the result of previous operations (If SUCCEEDED(hrPrev) equals false, no operation is executed.) *)
	END_VAR

END_FUNCTION

// Functions/Fourier Analysis/F_VN_CreateLowpassButterworthFilter

	{attribute 'TcIecLibraryType'}
	{attribute 'external_name' := 'F_VN_CreateLowpassButterworthFilter_GUID_DC88DEC8_1D01_574B_5355_192F6FE6DC63'}
	(* Creates a lowpass Butterworth filter, which can be applied to a frequency domain image by element-wise multiplication. *)
	FUNCTION F_VN_CreateLowpassButterworthFilter : HRESULT
	VAR_INPUT
		ipFilter	:	REFERENCE TO ITcVnImage;	(* Returns the created filter (1 channel of type REAL or LREAL, depending on bDoublePrecision. Non-zero interface pointers are reused.). *)
		nWidth	:	UDINT;	(* Filter width (even, >= 2, must match the width of the image it is applied to) *)
		nHeight	:	UDINT;	(* Filter height (even, >= 2, must match the height of the image it is applied to) *)
		bDoublePrecision	:	BOOL;	(* If true, the filter is generated with double precision (LREAL) instead of single precision (REAL). *)
		bOriginAtCenter	:	BOOL;	(* If true, the filter origin is shifted to the image center. *)
		fCutoffDistance	:	LREAL;	(* The cutoff distance of the Butterworth filter (> 0). *)
		nOrder	:	UDINT;	(* The order of the Butterworth filter (> 0). *)
		fScale	:	LREAL;	(* The scale factor of the Butterworth filter denominator term (> 0, e.g. 0.414 or 1.0). *)
		hrPrev	:	HRESULT;	(* HRESULT indicating the result of previous operations (If SUCCEEDED(hrPrev) equals false, no operation is executed.) *)
	END_VAR

END_FUNCTION

// Functions/Fourier Analysis/F_VN_CreateLowpassGaussianFilter

	{attribute 'TcIecLibraryType'}
	{attribute 'external_name' := 'F_VN_CreateLowpassGaussianFilter_GUID_178E14F4_2394_5970_703D_FDF316F7CE7D'}
	(* Creates a lowpass Gaussian filter, which can be applied to a frequency domain image by element-wise multiplication. *)
	FUNCTION F_VN_CreateLowpassGaussianFilter : HRESULT
	VAR_INPUT
		ipFilter	:	REFERENCE TO ITcVnImage;	(* Returns the created filter (1 channel of type REAL or LREAL, depending on bDoublePrecision. Non-zero interface pointers are reused.). *)
		nWidth	:	UDINT;	(* Filter width (even, >= 2, must match the width of the image it is applied to) *)
		nHeight	:	UDINT;	(* Filter height (even, >= 2, must match the height of the image it is applied to) *)
		bDoublePrecision	:	BOOL;	(* If true, the filter is generated with double precision (LREAL) instead of single precision (REAL). *)
		bOriginAtCenter	:	BOOL;	(* If true, the filter origin is shifted to the image center. *)
		fCutoffDistance	:	LREAL;	(* The cutoff distance of the Gaussian filter (> 0). *)
		hrPrev	:	HRESULT;	(* HRESULT indicating the result of previous operations (If SUCCEEDED(hrPrev) equals false, no operation is executed.) *)
	END_VAR

END_FUNCTION

// Functions/Fourier Analysis/F_VN_Dft

	{attribute 'TcIecLibraryType'}
	{attribute 'external_name' := 'F_VN_Dft_GUID_776AABF6_A102_5B49_7657_549B2A5BD382'}
	(* Computes the DFT for a given image. *)
	FUNCTION F_VN_Dft : HRESULT
	VAR_INPUT
		ipSpatialImage	:	ITcVnImage;	(* Source image (elements of type REAL or LREAL, 1 (Re) or 2 (Re + Im) channels) *)
		ipFrequencyImage	:	REFERENCE TO ITcVnImage;	(* Destination image (same type as ipSpatialImage, but number of channels and size can vary depending on bPackedCCS and bAutoPadding. *)
		bPackedCCS	:	BOOL;	(* If true and ipSpatialImage has only 1 channel, the result image will have 1 channel with packed complex-conjugate-symmetrical format results. Otherwise, the result image will have 2 separate channels (Re + Im), containing the full spectrum. *)
		bAutoPadding	:	BOOL;	(* If true, the input image is automatically padded (with 0s) to optimal size if required, to speed up dft (Creates a temporary copy so that ipSpatialImage content stays unchanged, which also requires some additional computation power. Therefore, it is recommended to compare execution times with and without padding.) *)
		hrPrev	:	HRESULT;	(* HRESULT indicating the result of previous operations (If SUCCEEDED(hrPrev) equals false, no operation is executed.) *)
	END_VAR

END_FUNCTION

// Functions/Fourier Analysis/F_VN_InverseDft

	{attribute 'TcIecLibraryType'}
	{attribute 'external_name' := 'F_VN_InverseDft_GUID_BA2889CE_1C85_5AF2_57A9_CC0F84CF6430'}
	(* Compute the inverse DFT for a given frequency image. *)
	FUNCTION F_VN_InverseDft : HRESULT
	VAR_INPUT
		ipFrequencyImage	:	ITcVnImage;	(* Source frequency image (elements of type REAL or LREAL, 1 (packed CCS) or 2 (Re + Im) channels) *)
		ipSpatialImage	:	REFERENCE TO ITcVnImage;	(* Destination image (Same type as ipFrequencyImage, but number of channels can vary depending on bRealOutput. An appropriate image will be created if required.) *)
		bRealOutput	:	BOOL;	(* Only relevant if ipFrequencyImage has 2 channels. If true, the result image will have only 1 channel. Otherwise, the result image will have 2 separate channels (Re + Im). If ipFrequencyImage has only 1 channel, packed CCS format is assumed and the result image will always have only 1 channel. *)
		hrPrev	:	HRESULT;	(* HRESULT indicating the result of previous operations (If SUCCEEDED(hrPrev) equals false, no operation is executed.) *)
	END_VAR

END_FUNCTION

// Functions/Fourier Analysis/F_VN_OptimalDftSize

	{attribute 'TcIecLibraryType'}
	{attribute 'external_name' := 'F_VN_OptimalDftSize_GUID_94CAE622_C038_5403_6D63_073A29300624'}
	(* Computes the optimal image size for applying a dft (can lead to better performance). *)
	FUNCTION F_VN_OptimalDftSize : HRESULT
	VAR_INPUT
		ipImage	:	ITcVnImage;	(* Source image for which to compute the optimal width and height *)
		nOptWidth	:	REFERENCE TO UDINT;	(* Returns the optimal width of the image *)
		nOptHeight	:	REFERENCE TO UDINT;	(* Returns the optimal height of the image *)
		hrPrev	:	HRESULT;	(* HRESULT indicating the result of previous operations (If SUCCEEDED(hrPrev) equals false, no operation is executed.) *)
	END_VAR

END_FUNCTION

// Functions/Fourier Analysis/F_VN_PadImageBorder

	{attribute 'TcIecLibraryType'}
	{attribute 'external_name' := 'F_VN_PadImageBorder_GUID_E9772FFB_3873_59D9_5182_A9F95598783B'}
	(* Add padding (zeros) around the original image borders. *)
	FUNCTION F_VN_PadImageBorder : HRESULT
	VAR_INPUT
		ipSrcImage	:	ITcVnImage;	(* Source image *)
		ipPaddedImage	:	REFERENCE TO ITcVnImage;	(* Padded destination image (Same type as ipSrcImage, an appropriate destination image will be created if required.) *)
		nTopBorder	:	UDINT;	(* Padding height in pixels above top border *)
		nBottomBorder	:	UDINT;	(* Padding height in pixels below bottom border *)
		nLeftBorder	:	UDINT;	(* Padding width in pixels before left border *)
		nRightBorder	:	UDINT;	(* Padding width in pixels after right border *)
		hrPrev	:	HRESULT;	(* HRESULT indicating the result of previous operations (If SUCCEEDED(hrPrev) equals false, no operation is executed.) *)
	END_VAR

END_FUNCTION

// Functions/Fourier Analysis/F_VN_PadImageBorderExp

	{attribute 'TcIecLibraryType'}
	{attribute 'external_name' := 'F_VN_PadImageBorderExp_GUID_4E5D984C_0EC6_5CFE_5340_5AEEED5A0A96'}
	(* Add padding around the original image borders. (expert function) *)
	FUNCTION F_VN_PadImageBorderExp : HRESULT
	VAR_INPUT
		ipSrcImage	:	ITcVnImage;	(* Source image *)
		ipPaddedImage	:	REFERENCE TO ITcVnImage;	(* Padded destination image (Same type as ipSrcImage, an appropriate destination image will be created if required.) *)
		nTopBorder	:	UDINT;	(* Padding height in pixels above top border *)
		nBottomBorder	:	UDINT;	(* Padding height in pixels below bottom border *)
		nLeftBorder	:	UDINT;	(* Padding width in pixels before left border *)
		nRightBorder	:	UDINT;	(* Padding width in pixels after right border *)
		ePaddingType	:	ETcVnBorderInterpolationMethod;	(* Specifies how the pixel values of the padding area are determined *)
		aPaddingValue	:	REFERENCE TO TcVnVector4_LREAL;	(* Specifies the padding value if CONSTANT is used *)
		hrPrev	:	HRESULT;	(* HRESULT indicating the result of previous operations (If SUCCEEDED(hrPrev) equals false, no operation is executed.) *)
	END_VAR

END_FUNCTION

// Functions/Drawing/F_VN_DrawCircle

	{attribute 'TcIecLibraryType'}
	{attribute 'external_name' := 'F_VN_DrawCircle_GUID_89161ACB_A0D2_54D2_5F15_07EFEA38DFF7'}
	(* Draws a circle. *)
	FUNCTION F_VN_DrawCircle : HRESULT
	VAR_INPUT
		nCenterX	:	UDINT;	(* x coordinate of the center *)
		nCenterY	:	UDINT;	(* y coordinate of the center *)
		nRadius	:	UDINT;	(* Radius *)
		ipDestImage	:	ITcVnImage;	(* Destination image *)
		aColor	:	REFERENCE TO TcVnVector4_LREAL;	(* Color *)
		nThickness	:	DINT;	(* Line thickness (if negative, the circle is filled) *)
		hrPrev	:	HRESULT;	(* HRESULT indicating the result of previous operations (If SUCCEEDED(hrPrev) equals false, no operation is executed.) *)
	END_VAR

END_FUNCTION

// Functions/Drawing/F_VN_DrawCircleExp

	{attribute 'TcIecLibraryType'}
	{attribute 'external_name' := 'F_VN_DrawCircleExp_GUID_87A92148_8E0F_5E76_7541_C7F9E4F45A40'}
	(* Draws a circle. *)
	FUNCTION F_VN_DrawCircleExp : HRESULT
	VAR_INPUT
		nCenterX	:	UDINT;	(* x coordinate of the center *)
		nCenterY	:	UDINT;	(* y coordinate of the center *)
		nRadius	:	UDINT;	(* Radius *)
		ipDestImage	:	ITcVnImage;	(* Destination image *)
		aColor	:	REFERENCE TO TcVnVector4_LREAL;	(* Color *)
		nThickness	:	DINT;	(* Line thickness (if negative, the circle is filled) *)
		eLineType	:	ETcVnLineType;	(* Line type *)
		hrPrev	:	HRESULT;	(* HRESULT indicating the result of previous operations (If SUCCEEDED(hrPrev) equals false, no operation is executed.) *)
	END_VAR

END_FUNCTION

// Functions/Drawing/F_VN_DrawCircles

	{attribute 'TcIecLibraryType'}
	{attribute 'external_name' := 'F_VN_DrawCircles_GUID_7FB211E7_35E7_5156_5B7A_2720C8A9B3EE'}
	(* Draws circles. *)
	FUNCTION F_VN_DrawCircles : HRESULT
	VAR_INPUT
		ipCircles	:	ITcVnContainer;	(* Container with circles (ContainerType_Vector_TcVnVector3_REAL; Each container element contains the x coordinate of the circle center [0], the y coordinate of the circle center [1], and the radius [2].) *)
		nCircleIndex	:	DINT;	(* Index of a specific circle to be drawn (if negative, all circles within the container are drawn) *)
		ipDestImage	:	ITcVnImage;	(* Destination image *)
		aColor	:	REFERENCE TO TcVnVector4_LREAL;	(* Color *)
		nThickness	:	DINT;	(* Line thickness (if negative, the circle is filled) *)
		hrPrev	:	HRESULT;	(* HRESULT indicating the result of previous operations (If SUCCEEDED(hrPrev) equals false, no operation is executed.) *)
	END_VAR

END_FUNCTION

// Functions/Drawing/F_VN_DrawCirclesExp

	{attribute 'TcIecLibraryType'}
	{attribute 'external_name' := 'F_VN_DrawCirclesExp_GUID_2CDC26EE_2BAC_5255_5EDF_F3B047AA1DF8'}
	(* Draws circles. (expert function) *)
	FUNCTION F_VN_DrawCirclesExp : HRESULT
	VAR_INPUT
		ipCircles	:	ITcVnContainer;	(* Container with circles (ContainerType_Vector_TcVnVector3_REAL; Each container element contains the x coordinate of the circle center [0], the y coordinate of the circle center [1], and the radius [2].) *)
		nCircleIndex	:	DINT;	(* Index of a specific circle to be drawn (if negative, all circles within the container are drawn) *)
		ipDestImage	:	ITcVnImage;	(* Destination image *)
		aColor	:	REFERENCE TO TcVnVector4_LREAL;	(* Color *)
		nThickness	:	DINT;	(* Line thickness (if negative, the circle is filled) *)
		eLineType	:	ETcVnLineType;	(* Line type *)
		hrPrev	:	HRESULT;	(* HRESULT indicating the result of previous operations (If SUCCEEDED(hrPrev) equals false, no operation is executed.) *)
	END_VAR

END_FUNCTION

// Functions/Drawing/F_VN_DrawCircularArc

	{attribute 'TcIecLibraryType'}
	{attribute 'external_name' := 'F_VN_DrawCircularArc_GUID_8E02D55A_1623_5005_4E1E_CDB49D77EA45'}
	(* Draws a circular arc. *)
	FUNCTION F_VN_DrawCircularArc : HRESULT
	VAR_INPUT
		stCircularArc	:	REFERENCE TO TcVnCircularArc;	(* Circular arc definition *)
		ipDestImage	:	ITcVnImage;	(* Destination image *)
		aColor	:	REFERENCE TO TcVnVector4_LREAL;	(* Color *)
		nThickness	:	DINT;	(* Line thickness (if negative, the arc is filled) *)
		hrPrev	:	HRESULT;	(* HRESULT indicating the result of previous operations (If SUCCEEDED(hrPrev) equals false, no operation is executed.) *)
	END_VAR

END_FUNCTION

// Functions/Drawing/F_VN_DrawCircularArcExp

	{attribute 'TcIecLibraryType'}
	{attribute 'external_name' := 'F_VN_DrawCircularArcExp_GUID_B5EB9E09_3F6C_5D4F_52AC_8168A629EE8B'}
	(* Draws a circular arc. (expert function) *)
	FUNCTION F_VN_DrawCircularArcExp : HRESULT
	VAR_INPUT
		stCircularArc	:	REFERENCE TO TcVnCircularArc;	(* Circular arc definition *)
		ipDestImage	:	ITcVnImage;	(* Destination image *)
		aColor	:	REFERENCE TO TcVnVector4_LREAL;	(* Color *)
		nThickness	:	DINT;	(* Line thickness (if negative, the arc is filled) *)
		eLineType	:	ETcVnLineType;	(* Line type *)
		hrPrev	:	HRESULT;	(* HRESULT indicating the result of previous operations (If SUCCEEDED(hrPrev) equals false, no operation is executed.) *)
	END_VAR

END_FUNCTION

// Functions/Drawing/F_VN_DrawContours

	{attribute 'TcIecLibraryType'}
	{attribute 'external_name' := 'F_VN_DrawContours_GUID_D1CE425A_8D05_501F_4F76_1DE7B8A03D5D'}
	(* Draws a single point set or multiple point sets that are interpreted as contours. *)
	FUNCTION F_VN_DrawContours : HRESULT
	VAR_INPUT
		ipContours	:	ITcVnContainer;	(* Single contour (ContainerType_Vector_TcVnPoint2_DINT) or multiple contours (ContainerType_Vector_Vector_TcVnPoint2_DINT) *)
		nContourIndex	:	DINT;	(* Index of a specific contour to be drawn (if negative, all contours within the container are drawn) *)
		ipDestImage	:	ITcVnImage;	(* Destination image *)
		aColor	:	REFERENCE TO TcVnVector4_LREAL;	(* Color *)
		nThickness	:	DINT;	(* Line thickness (if negative, the contours are filled) *)
		hrPrev	:	HRESULT;	(* HRESULT indicating the result of previous operations (If SUCCEEDED(hrPrev) equals false, no operation is executed.) *)
	END_VAR

END_FUNCTION

// Functions/Drawing/F_VN_DrawContoursExp

	{attribute 'TcIecLibraryType'}
	{attribute 'external_name' := 'F_VN_DrawContoursExp_GUID_A2A3129F_3E44_54FD_53E3_9AFA80881185'}
	(* Draws a single point set or multiple point sets that are interpreted as contours. (expert function) *)
	FUNCTION F_VN_DrawContoursExp : HRESULT
	VAR_INPUT
		ipContours	:	ITcVnContainer;	(* Single contour (ContainerType_Vector_TcVnPoint2_DINT) or multiple contours (ContainerType_Vector_Vector_TcVnPoint2_DINT) *)
		nContourIndex	:	DINT;	(* Index of a specific contour to be drawn (if negative, all contours within the container are drawn) *)
		ipDestImage	:	ITcVnImage;	(* Destination image *)
		aColor	:	REFERENCE TO TcVnVector4_LREAL;	(* Color *)
		nThickness	:	DINT;	(* Line thickness (if negative, the contours are filled) *)
		eLineType	:	ETcVnLineType;	(* Line type *)
		ipHierarchy	:	ITcVnContainer;	(* Contour hierarchy (ContainerType_Vector_TcVnVector4_DINT) *)
		nMaxLevel	:	DINT;	(* Maximum level of contours to be drawn *)
		aOffset	:	REFERENCE TO TcVnPoint;	(* Offset by which every contour point is shifted *)
		hrPrev	:	HRESULT;	(* HRESULT indicating the result of previous operations (If SUCCEEDED(hrPrev) equals false, no operation is executed.) *)
	END_VAR

END_FUNCTION

// Functions/Drawing/F_VN_DrawEllipse

	{attribute 'TcIecLibraryType'}
	{attribute 'external_name' := 'F_VN_DrawEllipse_GUID_58D3EC1D_08E9_5FDA_5852_FE65F7766D0F'}
	(* Draws an ellipse. *)
	FUNCTION F_VN_DrawEllipse : HRESULT
	VAR_INPUT
		stEllipse	:	REFERENCE TO TcVnRotatedRectangle;	(* Ellipse to be drawn (rotation angle in degrees) *)
		ipDestImage	:	ITcVnImage;	(* Destination image *)
		aColor	:	REFERENCE TO TcVnVector4_LREAL;	(* Color *)
		nThickness	:	DINT;	(* Line thickness (if negative, the ellipse is filled) *)
		hrPrev	:	HRESULT;	(* HRESULT indicating the result of previous operations (If SUCCEEDED(hrPrev) equals false, no operation is executed.) *)
	END_VAR

END_FUNCTION

// Functions/Drawing/F_VN_DrawEllipseExp

	{attribute 'TcIecLibraryType'}
	{attribute 'external_name' := 'F_VN_DrawEllipseExp_GUID_A9DF7C51_CADF_59B2_7E65_A029AE7706DF'}
	(* Draws an ellipse. (expert function) *)
	FUNCTION F_VN_DrawEllipseExp : HRESULT
	VAR_INPUT
		stEllipse	:	REFERENCE TO TcVnRotatedRectangle;	(* Ellipse to be drawn (rotation angle in degrees) *)
		ipDestImage	:	ITcVnImage;	(* Destination image *)
		aColor	:	REFERENCE TO TcVnVector4_LREAL;	(* Color *)
		nThickness	:	DINT;	(* Line thickness (if negative, the ellipse is filled) *)
		eLineType	:	ETcVnLineType;	(* Line type *)
		hrPrev	:	HRESULT;	(* HRESULT indicating the result of previous operations (If SUCCEEDED(hrPrev) equals false, no operation is executed.) *)
	END_VAR

END_FUNCTION

// Functions/Drawing/F_VN_DrawKeypoints

	{attribute 'TcIecLibraryType'}
	{attribute 'external_name' := 'F_VN_DrawKeypoints_GUID_1080A168_C4CC_5BC7_50E0_5D55F011CDF1'}
	(* Draws the keypoints for visualization purpose. *)
	FUNCTION F_VN_DrawKeypoints : HRESULT
	VAR_INPUT
		ipSrcImage	:	ITcVnImage;	(* Source image (elements of type USINT) *)
		ipKeyPoints	:	ITcVnContainer;	(* Container with the keypoints (ContainerType_Vector_TcVnKeyPoint) *)
		ipDestImage	:	REFERENCE TO ITcVnImage;	(* Destination image (An appropriate image will be created if required.) *)
		hrPrev	:	HRESULT;	(* HRESULT indicating the result of previous operations (If SUCCEEDED(hrPrev) equals false, no operation is executed.) *)
	END_VAR

END_FUNCTION

// Functions/Drawing/F_VN_DrawKeypointsExp

	{attribute 'TcIecLibraryType'}
	{attribute 'external_name' := 'F_VN_DrawKeypointsExp_GUID_BEAB2C06_7266_5B04_6D10_85ED06B16666'}
	(* Draws the keypoints for visualization purpose. (expert function) *)
	FUNCTION F_VN_DrawKeypointsExp : HRESULT
	VAR_INPUT
		ipSrcImage	:	ITcVnImage;	(* Source image (elements of type USINT) *)
		ipKeyPoints	:	ITcVnContainer;	(* Container with the keypoints (ContainerType_Vector_TcVnKeyPoint) *)
		ipDestImage	:	REFERENCE TO ITcVnImage;	(* Destination image (An appropriate image will be created if required.) *)
		aColor	:	REFERENCE TO TcVnVector4_LREAL;	(* Color to draw the keypoints (for {-1, -1, -1, -1}, a random color is chosen for each point) *)
		eFlags	:	ETcVnDrawMatchesFlags;	(* A combination of flags to support overdrawing an existing destination image and/or drawing additional (Rich-)Keypoint information (size and orientation) *)
		hrPrev	:	HRESULT;	(* HRESULT indicating the result of previous operations (If SUCCEEDED(hrPrev) equals false, no operation is executed.) *)
	END_VAR

END_FUNCTION

// Functions/Drawing/F_VN_DrawLine

	{attribute 'TcIecLibraryType'}
	{attribute 'external_name' := 'F_VN_DrawLine_GUID_6E28C4B1_0F97_510D_6B83_C04C0B5D97F9'}
	(* Draws a line. *)
	FUNCTION F_VN_DrawLine : HRESULT
	VAR_INPUT
		nX1	:	UDINT;	(* x coordinate of the start point *)
		nY1	:	UDINT;	(* y coordinate of the start point *)
		nX2	:	UDINT;	(* x coordinate of the end point *)
		nY2	:	UDINT;	(* y coordinate of the end point *)
		ipDestImage	:	ITcVnImage;	(* Destination image *)
		aColor	:	REFERENCE TO TcVnVector4_LREAL;	(* Color *)
		nThickness	:	DINT;	(* Line thickness *)
		hrPrev	:	HRESULT;	(* HRESULT indicating the result of previous operations (If SUCCEEDED(hrPrev) equals false, no operation is executed.) *)
	END_VAR

END_FUNCTION

// Functions/Drawing/F_VN_DrawLineExp

	{attribute 'TcIecLibraryType'}
	{attribute 'external_name' := 'F_VN_DrawLineExp_GUID_36788353_26FE_522E_4610_D7DDF0C11D62'}
	(* Draws a line. (expert function) *)
	FUNCTION F_VN_DrawLineExp : HRESULT
	VAR_INPUT
		nX1	:	UDINT;	(* x coordinate of the start point *)
		nY1	:	UDINT;	(* y coordinate of the start point *)
		nX2	:	UDINT;	(* x coordinate of the end point *)
		nY2	:	UDINT;	(* y coordinate of the end point *)
		ipDestImage	:	ITcVnImage;	(* Destination image *)
		aColor	:	REFERENCE TO TcVnVector4_LREAL;	(* Color *)
		nThickness	:	DINT;	(* Line thickness *)
		eLineType	:	ETcVnLineType;	(* Line type *)
		nShift	:	UDINT;	(* Fractional bits of the coordinates (bit shift) *)
		hrPrev	:	HRESULT;	(* HRESULT indicating the result of previous operations (If SUCCEEDED(hrPrev) equals false, no operation is executed.) *)
	END_VAR

END_FUNCTION

// Functions/Drawing/F_VN_DrawLine_TcVnVector4_DINT

	{attribute 'TcIecLibraryType'}
	{attribute 'external_name' := 'F_VN_DrawLine_TcVnVector4_DINT_GUID_E072396A_AF24_5219_6AA7_BFD408437599'}
	(* Draws a line. *)
	FUNCTION F_VN_DrawLine_TcVnVector4_DINT : HRESULT
	VAR_INPUT
		aLine	:	REFERENCE TO TcVnVector4_DINT;	(* The start and end point of a line segment [x1, y1, x2, y2] *)
		ipDestImage	:	ITcVnImage;	(* Destination image *)
		aColor	:	REFERENCE TO TcVnVector4_LREAL;	(* Color *)
		nThickness	:	DINT;	(* Line thickness *)
		hrPrev	:	HRESULT;	(* HRESULT indicating the result of previous operations (If SUCCEEDED(hrPrev) equals false, no operation is executed.) *)
	END_VAR

END_FUNCTION

// Functions/Drawing/F_VN_DrawLineExp_TcVnVector4_DINT

	{attribute 'TcIecLibraryType'}
	{attribute 'external_name' := 'F_VN_DrawLineExp_TcVnVector4_DINT_GUID_801C6446_4A7E_5A55_669E_B3FED405229F'}
	(* Draws a line. (expert function) *)
	FUNCTION F_VN_DrawLineExp_TcVnVector4_DINT : HRESULT
	VAR_INPUT
		aLine	:	REFERENCE TO TcVnVector4_DINT;	(* The start and end point of a line segment [x1, y1, x2, y2] *)
		ipDestImage	:	ITcVnImage;	(* Destination image *)
		aColor	:	REFERENCE TO TcVnVector4_LREAL;	(* Color *)
		nThickness	:	DINT;	(* Line thickness *)
		eLineType	:	ETcVnLineType;	(* Line type *)
		nShift	:	UDINT;	(* Fractional bits of the coordinates (bit shift) *)
		hrPrev	:	HRESULT;	(* HRESULT indicating the result of previous operations (If SUCCEEDED(hrPrev) equals false, no operation is executed.) *)
	END_VAR

END_FUNCTION

// Functions/Drawing/F_VN_DrawLine_TcVnVector4_LREAL

	{attribute 'TcIecLibraryType'}
	{attribute 'external_name' := 'F_VN_DrawLine_TcVnVector4_LREAL_GUID_1BAC7196_286C_5BDF_51AF_4B98EE8C297C'}
	(* Draws a line. *)
	FUNCTION F_VN_DrawLine_TcVnVector4_LREAL : HRESULT
	VAR_INPUT
		aLine	:	REFERENCE TO TcVnVector4_LREAL;	(* The first and second element describe the x and y component of the direction vector. The third and fourth element describe the x and y component of the position vector. *)
		ipDestImage	:	ITcVnImage;	(* Destination image *)
		aColor	:	REFERENCE TO TcVnVector4_LREAL;	(* Color *)
		nThickness	:	DINT;	(* Line thickness *)
		hrPrev	:	HRESULT;	(* HRESULT indicating the result of previous operations (If SUCCEEDED(hrPrev) equals false, no operation is executed.) *)
	END_VAR

END_FUNCTION

// Functions/Drawing/F_VN_DrawLineExp_TcVnVector4_LREAL

	{attribute 'TcIecLibraryType'}
	{attribute 'external_name' := 'F_VN_DrawLineExp_TcVnVector4_LREAL_GUID_A2C56657_DB83_5AE9_52E6_8F7A26B87271'}
	(* Draws a line. (expert function) *)
	FUNCTION F_VN_DrawLineExp_TcVnVector4_LREAL : HRESULT
	VAR_INPUT
		aLine	:	REFERENCE TO TcVnVector4_LREAL;	(* The first and second element describe the x and y component of the direction vector. The third and fourth element describe the x and y component of the position vector. *)
		ipDestImage	:	ITcVnImage;	(* Destination image *)
		aColor	:	REFERENCE TO TcVnVector4_LREAL;	(* Color *)
		nThickness	:	DINT;	(* Line thickness *)
		eLineType	:	ETcVnLineType;	(* Line type *)
		nShift	:	UDINT;	(* Fractional bits of the coordinates (bit shift) *)
		hrPrev	:	HRESULT;	(* HRESULT indicating the result of previous operations (If SUCCEEDED(hrPrev) equals false, no operation is executed.) *)
	END_VAR

END_FUNCTION

// Functions/Drawing/F_VN_DrawLines

	{attribute 'TcIecLibraryType'}
	{attribute 'external_name' := 'F_VN_DrawLines_GUID_944FB242_F673_5A26_54D6_A40E05AC1154'}
	(* Draws lines. *)
	FUNCTION F_VN_DrawLines : HRESULT
	VAR_INPUT
		ipLines	:	ITcVnContainer;	(* Container with line descriptions (ContainerType_Vector_TcVnVector2_REAL: the distance from the origin [0] in pixels and the rotation angle [1] in radians. ContainerType_Vector_TcVnVector4_LREAL: the first and second element describe the x and y component of a vector collinear to the line. The third and fourth element describe the x and y component of a point on the line. ContainerType_Vector_TcVnVector4_DINT: start and end point [x1, y1, x2, y2]) *)
		nLineIndex	:	DINT;	(* Index of a specific line to be drawn (if negative, all lines within the container are drawn) *)
		ipDestImage	:	ITcVnImage;	(* Destination image *)
		aColor	:	REFERENCE TO TcVnVector4_LREAL;	(* Color *)
		nThickness	:	DINT;	(* Line thickness *)
		hrPrev	:	HRESULT;	(* HRESULT indicating the result of previous operations (If SUCCEEDED(hrPrev) equals false, no operation is executed.) *)
	END_VAR

END_FUNCTION

// Functions/Drawing/F_VN_DrawLinesExp

	{attribute 'TcIecLibraryType'}
	{attribute 'external_name' := 'F_VN_DrawLinesExp_GUID_AF5C1299_A9CD_5B71_44A7_2BD74C459A66'}
	(* Draws lines. (expert function) *)
	FUNCTION F_VN_DrawLinesExp : HRESULT
	VAR_INPUT
		ipLines	:	ITcVnContainer;	(* Container with line descriptions (ContainerType_Vector_TcVnVector2_REAL: the distance from the origin [0] in pixels and the rotation angle [1] in radians. ContainerType_Vector_TcVnVector4_LREAL: the first and second element describe the x and y component of a vector collinear to the line. The third and fourth element describe the x and y component of a point on the line. ContainerType_Vector_TcVnVector4_DINT: start and end point [x1, y1, x2, y2]) *)
		nLineIndex	:	DINT;	(* Index of a specific line to be drawn (if negative, all lines within the container are drawn) *)
		ipDestImage	:	ITcVnImage;	(* Destination image *)
		aColor	:	REFERENCE TO TcVnVector4_LREAL;	(* Color *)
		nThickness	:	DINT;	(* Line thickness *)
		eLineType	:	ETcVnLineType;	(* Line type *)
		nShift	:	UDINT;	(* Fractional bits of the coordinates (bit shift) *)
		hrPrev	:	HRESULT;	(* HRESULT indicating the result of previous operations (If SUCCEEDED(hrPrev) equals false, no operation is executed.) *)
	END_VAR

END_FUNCTION

// Functions/Drawing/F_VN_DrawMatches

	{attribute 'TcIecLibraryType'}
	{attribute 'external_name' := 'F_VN_DrawMatches_GUID_7F929F05_4897_5BBB_7E32_965C505EB4AE'}
	(* Draws the keypoints and matches for visualization purpose. *)
	FUNCTION F_VN_DrawMatches : HRESULT
	VAR_INPUT
		ipSrcImage1	:	ITcVnImage;	(* Source image 1 (elements of type USINT) *)
		ipKeyPoints1	:	ITcVnContainer;	(* Container with the keypoints 1 (ContainerType_Vector_TcVnKeyPoint) *)
		ipSrcImage2	:	ITcVnImage;	(* Source image 2 (elements of type USINT) *)
		ipKeyPoints2	:	ITcVnContainer;	(* Container with the keypoints 2 (ContainerType_Vector_TcVnKeyPoint) *)
		ipMatches1To2	:	ITcVnContainer;	(* Container with the descriptor matches (ContainerType_Vector_TcVnDMatch) *)
		ipDestImage	:	REFERENCE TO ITcVnImage;	(* Destination image (An appropriate image will be created if required.) *)
		hrPrev	:	HRESULT;	(* HRESULT indicating the result of previous operations (If SUCCEEDED(hrPrev) equals false, no operation is executed.) *)
	END_VAR

END_FUNCTION

// Functions/Drawing/F_VN_DrawMatchesExp

	{attribute 'TcIecLibraryType'}
	{attribute 'external_name' := 'F_VN_DrawMatchesExp_GUID_352BFE6D_CECC_5B6B_66D9_C393D0493835'}
	(* Draws the keypoints and matches for visualization purpose. (expert function) *)
	FUNCTION F_VN_DrawMatchesExp : HRESULT
	VAR_INPUT
		ipSrcImage1	:	ITcVnImage;	(* Source image 1 (elements of type USINT) *)
		ipKeyPoints1	:	ITcVnContainer;	(* Container with the keypoints 1 (ContainerType_Vector_TcVnKeyPoint) *)
		ipSrcImage2	:	ITcVnImage;	(* Source image 2 (elements of type USINT) *)
		ipKeyPoints2	:	ITcVnContainer;	(* Container with the keypoints 2 (ContainerType_Vector_TcVnKeyPoint) *)
		ipMatches1To2	:	ITcVnContainer;	(* Container with the descriptor matches (ContainerType_Vector_TcVnDMatch) *)
		ipDestImage	:	REFERENCE TO ITcVnImage;	(* Destination image (An appropriate image will be created if required.) *)
		aMatchColor	:	REFERENCE TO TcVnVector4_LREAL;	(* Color to draw the matches (for {-1, -1, -1, -1}, a random color is chosen for each point and line) *)
		aSingleColor	:	REFERENCE TO TcVnVector4_LREAL;	(* Color to draw the single keypoints (for {-1, -1, -1, -1}, a random color is chosen for each point) *)
		ipMatchesMask	:	ITcVnContainer;	(* Mask to select the matches to be drawn (ContainerType_Vector_SINT; Set to 0 if all matches should be drawn.) *)
		eFlags	:	ETcVnDrawMatchesFlags;	(* A combination of flags to support overdrawing an existing destination image and/or drawing additional (Rich-)Keypoint information (size and orientation) and/or skipping single keypoints *)
		hrPrev	:	HRESULT;	(* HRESULT indicating the result of previous operations (If SUCCEEDED(hrPrev) equals false, no operation is executed.) *)
	END_VAR

END_FUNCTION

// Functions/Drawing/F_VN_DrawPoint

	{attribute 'TcIecLibraryType'}
	{attribute 'external_name' := 'F_VN_DrawPoint_GUID_18AC8FCB_3946_5DF8_44E6_A1A2C5AED46D'}
	(* Draws a point. *)
	FUNCTION F_VN_DrawPoint : HRESULT
	VAR_INPUT
		nX	:	UDINT;	(* x coordinate of the point *)
		nY	:	UDINT;	(* y coordinate of the point *)
		ipDestImage	:	ITcVnImage;	(* Destination image *)
		eShape	:	ETcVnDrawShape;	(* Point shape *)
		aColor	:	REFERENCE TO TcVnVector4_LREAL;	(* Color *)
		hrPrev	:	HRESULT;	(* HRESULT indicating the result of previous operations (If SUCCEEDED(hrPrev) equals false, no operation is executed.) *)
	END_VAR

END_FUNCTION

// Functions/Drawing/F_VN_DrawPointExp

	{attribute 'TcIecLibraryType'}
	{attribute 'external_name' := 'F_VN_DrawPointExp_GUID_FF041B97_57AF_5442_7BF9_99A69F7B19DE'}
	(* Draw a point. (expert function) *)
	FUNCTION F_VN_DrawPointExp : HRESULT
	VAR_INPUT
		nX	:	UDINT;	(* x coordinate of the point *)
		nY	:	UDINT;	(* y coordinate of the point *)
		ipDestImage	:	ITcVnImage;	(* Destination image *)
		eShape	:	ETcVnDrawShape;	(* Point shape *)
		aColor	:	REFERENCE TO TcVnVector4_LREAL;	(* Color *)
		nSize	:	UDINT;	(* Size of the shape (half width) *)
		nThickness	:	DINT;	(* Line thickness (if negative, the shape is filled if it is closed) *)
		eLineType	:	ETcVnLineType;	(* Line type *)
		hrPrev	:	HRESULT;	(* HRESULT indicating the result of previous operations (If SUCCEEDED(hrPrev) equals false, no operation is executed.) *)
	END_VAR

END_FUNCTION

// Functions/Drawing/F_VN_DrawPoints

	{attribute 'TcIecLibraryType'}
	{attribute 'external_name' := 'F_VN_DrawPoints_GUID_157DCD8E_5B70_54A0_6D53_4F015496D56C'}
	(* Draw a collection of points. *)
	FUNCTION F_VN_DrawPoints : HRESULT
	VAR_INPUT
		ipPoints	:	ITcVnContainer;	(* Container with TcVnPoint2_DINT or TcVnPoint2_REAL elements *)
		ipDestImage	:	ITcVnImage;	(* Destination image *)
		eShape	:	ETcVnDrawShape;	(* Point shape *)
		aColor	:	REFERENCE TO TcVnVector4_LREAL;	(* Color *)
		hrPrev	:	HRESULT;	(* HRESULT indicating the result of previous operations (If SUCCEEDED(hrPrev) equals false, no operation is executed.) *)
	END_VAR

END_FUNCTION

// Functions/Drawing/F_VN_DrawPointsExp

	{attribute 'TcIecLibraryType'}
	{attribute 'external_name' := 'F_VN_DrawPointsExp_GUID_C707625A_54FB_56DE_7DA1_AEED948C8BA5'}
	(* Draw a collection of points. (expert function) *)
	FUNCTION F_VN_DrawPointsExp : HRESULT
	VAR_INPUT
		ipPoints	:	ITcVnContainer;	(* Container with TcVnPoint2_DINT or TcVnPoint2_REAL elements *)
		ipDestImage	:	ITcVnImage;	(* Destination image *)
		eShape	:	ETcVnDrawShape;	(* Point shape *)
		aColor	:	REFERENCE TO TcVnVector4_LREAL;	(* Color *)
		nSize	:	UDINT;	(* Size of the shape (half width) *)
		nThickness	:	DINT;	(* Line thickness (if negative, the shape is filled if it is closed) *)
		eLineType	:	ETcVnLineType;	(* Line type *)
		hrPrev	:	HRESULT;	(* HRESULT indicating the result of previous operations (If SUCCEEDED(hrPrev) equals false, no operation is executed.) *)
	END_VAR

END_FUNCTION

// Functions/Drawing/F_VN_DrawRectangle

	{attribute 'TcIecLibraryType'}
	{attribute 'external_name' := 'F_VN_DrawRectangle_GUID_39C3D5AC_1776_54A5_6124_C5C4FB97827A'}
	(* Draw a rectangle. *)
	FUNCTION F_VN_DrawRectangle : HRESULT
	VAR_INPUT
		nTopLeftX	:	UDINT;	(* x coordinate of the top left corner *)
		nTopLeftY	:	UDINT;	(* y coordinate of the top left corner *)
		nBottomRightX	:	UDINT;	(* x coordinate of the bottom right corner *)
		nBottomRightY	:	UDINT;	(* y coordinate of the bottom right corner *)
		ipDestImage	:	ITcVnImage;	(* Destination image *)
		aColor	:	REFERENCE TO TcVnVector4_LREAL;	(* Color *)
		nThickness	:	DINT;	(* Line thickness (if negative, the rectangle is filled) *)
		hrPrev	:	HRESULT;	(* HRESULT indicating the result of previous operations (If SUCCEEDED(hrPrev) equals false, no operation is executed.) *)
	END_VAR

END_FUNCTION

// Functions/Drawing/F_VN_DrawRectangle_TcVnRectangle_UDINT

	{attribute 'TcIecLibraryType'}
	{attribute 'external_name' := 'F_VN_DrawRectangle_TcVnRectangle_UDINT_GUID_B8C7F099_6306_5617_5FEB_2F881CD12756'}
	(* Draw a rectangle. *)
	FUNCTION F_VN_DrawRectangle_TcVnRectangle_UDINT : HRESULT
	VAR_INPUT
		stRectangle	:	REFERENCE TO TcVnRectangle_UDINT;	(* Rectangle to be drawn *)
		ipDestImage	:	ITcVnImage;	(* Destination image *)
		aColor	:	REFERENCE TO TcVnVector4_LREAL;	(* Color *)
		nThickness	:	DINT;	(* Line thickness (if negative, the rectangle is filled) *)
		hrPrev	:	HRESULT;	(* HRESULT indicating the result of previous operations (If SUCCEEDED(hrPrev) equals false, no operation is executed.) *)
	END_VAR

END_FUNCTION

// Functions/Drawing/F_VN_DrawRotatedRectangle

	{attribute 'TcIecLibraryType'}
	{attribute 'external_name' := 'F_VN_DrawRotatedRectangle_GUID_1AAA129B_D238_5001_6F30_4A31098E55D9'}
	(* Draw a rectangle. *)
	FUNCTION F_VN_DrawRotatedRectangle : HRESULT
	VAR_INPUT
		stRectangle	:	REFERENCE TO TcVnRotatedRectangle;	(* Rectangle to be drawn (rotation angle in degrees) *)
		ipDestImage	:	ITcVnImage;	(* Destination image *)
		aColor	:	REFERENCE TO TcVnVector4_LREAL;	(* Color *)
		nThickness	:	DINT;	(* Line thickness (if negative, the rectangle is filled) *)
		hrPrev	:	HRESULT;	(* HRESULT indicating the result of previous operations (If SUCCEEDED(hrPrev) equals false, no operation is executed.) *)
	END_VAR

END_FUNCTION

// Functions/Drawing/F_VN_DrawRotatedRectangleExp

	{attribute 'TcIecLibraryType'}
	{attribute 'external_name' := 'F_VN_DrawRotatedRectangleExp_GUID_0DB33F1E_2A29_5DFC_648F_69B8715D350D'}
	(* Draw a rectangle. (expert function) *)
	FUNCTION F_VN_DrawRotatedRectangleExp : HRESULT
	VAR_INPUT
		stRectangle	:	REFERENCE TO TcVnRotatedRectangle;	(* Rectangle to be drawn (rotation angle in degrees) *)
		ipDestImage	:	ITcVnImage;	(* Destination image *)
		aColor	:	REFERENCE TO TcVnVector4_LREAL;	(* Color *)
		nThickness	:	DINT;	(* Line thickness (if negative, the rectangle is filled) *)
		eLineType	:	ETcVnLineType;	(* Line type *)
		hrPrev	:	HRESULT;	(* HRESULT indicating the result of previous operations (If SUCCEEDED(hrPrev) equals false, no operation is executed.) *)
	END_VAR

END_FUNCTION

// Functions/Drawing/F_VN_FillCircle

	{attribute 'TcIecLibraryType'}
	{attribute 'external_name' := 'F_VN_FillCircle_GUID_A442D3C0_571C_5491_5C49_944661219EBF'}
	(* Paint a filled circle. *)
	FUNCTION F_VN_FillCircle : HRESULT
	VAR_INPUT
		nCenterX	:	UDINT;	(* x coordinate of the center *)
		nCenterY	:	UDINT;	(* y coordinate of the center *)
		nRadius	:	UDINT;	(* Radius *)
		ipDestImage	:	ITcVnImage;	(* Destination image *)
		aColor	:	REFERENCE TO TcVnVector4_LREAL;	(* Color *)
		hrPrev	:	HRESULT;	(* HRESULT indicating the result of previous operations (If SUCCEEDED(hrPrev) equals false, no operation is executed.) *)
	END_VAR

END_FUNCTION

// Functions/Drawing/F_VN_FillContours

	{attribute 'TcIecLibraryType'}
	{attribute 'external_name' := 'F_VN_FillContours_GUID_69A220E8_B575_5AB4_6E9F_3F0E9FDD958C'}
	(* Paint a single point set or multiple point sets that are interpreted as contours. *)
	FUNCTION F_VN_FillContours : HRESULT
	VAR_INPUT
		ipContours	:	ITcVnContainer;	(* Single contour (ContainerType_Vector_TcVnPoint2_DINT) or multiple contours (ContainerType_Vector_Vector_TcVnPoint2_DINT) *)
		nContourIndex	:	DINT;	(* Index of a specific contour to be drawn (if negative, all contours within the container are drawn) *)
		ipDestImage	:	ITcVnImage;	(* Destination image *)
		aColor	:	REFERENCE TO TcVnVector4_LREAL;	(* Color *)
		hrPrev	:	HRESULT;	(* HRESULT indicating the result of previous operations (If SUCCEEDED(hrPrev) equals false, no operation is executed.) *)
	END_VAR

END_FUNCTION

// Functions/Drawing/F_VN_FillEllipse

	{attribute 'TcIecLibraryType'}
	{attribute 'external_name' := 'F_VN_FillEllipse_GUID_AF6C6834_3867_511E_65E6_34DFC653C086'}
	(* Paint a filled ellipse. *)
	FUNCTION F_VN_FillEllipse : HRESULT
	VAR_INPUT
		stEllipse	:	REFERENCE TO TcVnRotatedRectangle;	(* Ellipse to be painted (rotation angle in degrees) *)
		ipDestImage	:	ITcVnImage;	(* Destination image *)
		aColor	:	REFERENCE TO TcVnVector4_LREAL;	(* Color *)
		hrPrev	:	HRESULT;	(* HRESULT indicating the result of previous operations (If SUCCEEDED(hrPrev) equals false, no operation is executed.) *)
	END_VAR

END_FUNCTION

// Functions/Drawing/F_VN_FillRectangle

	{attribute 'TcIecLibraryType'}
	{attribute 'external_name' := 'F_VN_FillRectangle_GUID_4543B41A_EEDB_54F3_5955_277DD0B1F8BF'}
	(* Paint a filled rectangle. *)
	FUNCTION F_VN_FillRectangle : HRESULT
	VAR_INPUT
		nTopLeftX	:	UDINT;	(* x coordinate of the top left corner *)
		nTopLeftY	:	UDINT;	(* y coordinate of the top left corner *)
		nBottomRightX	:	UDINT;	(* x coordinate of the bottom right corner *)
		nBottomRightY	:	UDINT;	(* y coordinate of the bottom right corner *)
		ipDestImage	:	ITcVnImage;	(* Destination image *)
		aColor	:	REFERENCE TO TcVnVector4_LREAL;	(* Color *)
		hrPrev	:	HRESULT;	(* HRESULT indicating the result of previous operations (If SUCCEEDED(hrPrev) equals false, no operation is executed.) *)
	END_VAR

END_FUNCTION

// Functions/Drawing/F_VN_FillRotatedRectangle

	{attribute 'TcIecLibraryType'}
	{attribute 'external_name' := 'F_VN_FillRotatedRectangle_GUID_F6AE6BFA_E696_5610_6566_802FD5D065A8'}
	(* Paint a filled rectangle. *)
	FUNCTION F_VN_FillRotatedRectangle : HRESULT
	VAR_INPUT
		stRectangle	:	REFERENCE TO TcVnRotatedRectangle;	(* Rectangle to be painted (rotation angle in degrees) *)
		ipDestImage	:	ITcVnImage;	(* Destination image *)
		aColor	:	REFERENCE TO TcVnVector4_LREAL;	(* Color *)
		hrPrev	:	HRESULT;	(* HRESULT indicating the result of previous operations (If SUCCEEDED(hrPrev) equals false, no operation is executed.) *)
	END_VAR

END_FUNCTION

// Functions/Drawing/F_VN_PutLabel

	{attribute 'TcIecLibraryType'}
	{attribute 'external_name' := 'F_VN_PutLabel_GUID_5F94C54B_EE19_55F4_6015_4F59363F04AA'}
	(* Write a label (black text on white background) into an image. *)
	FUNCTION F_VN_PutLabel : HRESULT
	VAR_IN_OUT CONSTANT
		sText	:	STRING;	(* Text *)
	END_VAR
	VAR_INPUT
		ipDestImage	:	ITcVnImage;	(* Destination image *)
		nX	:	UDINT;	(* x coordinate (bottom left) *)
		nY	:	UDINT;	(* y coordinate (bottom left) *)
		fFontScale	:	LREAL;	(* Scaling factor *)
		hrPrev	:	HRESULT;	(* HRESULT indicating the result of previous operations (If SUCCEEDED(hrPrev) equals false, no operation is executed.) *)
	END_VAR

END_FUNCTION

// Functions/Drawing/F_VN_PutLabelExp

	{attribute 'TcIecLibraryType'}
	{attribute 'external_name' := 'F_VN_PutLabelExp_GUID_D160A5E8_28E2_5474_4698_1A2E933B02E9'}
	(* Write a label (text on unified background) into an image. (expert function) *)
	FUNCTION F_VN_PutLabelExp : HRESULT
	VAR_IN_OUT CONSTANT
		sText	:	STRING;	(* Text *)
	END_VAR
	VAR_INPUT
		ipDestImage	:	ITcVnImage;	(* Destination image *)
		nX	:	UDINT;	(* x coordinate (bottom left) *)
		nY	:	UDINT;	(* y coordinate (bottom left) *)
		fFontScale	:	LREAL;	(* Scaling factor *)
		nThickness	:	UDINT;	(* Line thickness *)
		eFontType	:	ETcVnFontType;	(* Font type *)
		aFontColor	:	REFERENCE TO TcVnVector4_LREAL;	(* Font color *)
		aBackgroundColor	:	REFERENCE TO TcVnVector4_LREAL;	(* Background color *)
		eLineType	:	ETcVnLineType;	(* Line type *)
		hrPrev	:	HRESULT;	(* HRESULT indicating the result of previous operations (If SUCCEEDED(hrPrev) equals false, no operation is executed.) *)
	END_VAR

END_FUNCTION

// Functions/Drawing/F_VN_PutText

	{attribute 'TcIecLibraryType'}
	{attribute 'external_name' := 'F_VN_PutText_GUID_79318EA1_21BF_5AAA_61CB_A09C5E581FAA'}
	(* Write text into an image. *)
	FUNCTION F_VN_PutText : HRESULT
	VAR_IN_OUT CONSTANT
		sText	:	STRING;	(* Text *)
	END_VAR
	VAR_INPUT
		ipDestImage	:	ITcVnImage;	(* Destination image *)
		nX	:	UDINT;	(* x coordinate (bottom left) *)
		nY	:	UDINT;	(* y coordinate (bottom left) *)
		eFontType	:	ETcVnFontType;	(* Font type *)
		fFontScale	:	LREAL;	(* Scaling factor *)
		aColor	:	REFERENCE TO TcVnVector4_LREAL;	(* Text color *)
		hrPrev	:	HRESULT;	(* HRESULT indicating the result of previous operations (If SUCCEEDED(hrPrev) equals false, no operation is executed.) *)
	END_VAR

END_FUNCTION

// Functions/Drawing/F_VN_PutTextExp

	{attribute 'TcIecLibraryType'}
	{attribute 'external_name' := 'F_VN_PutTextExp_GUID_2B38E426_431D_547D_5DA1_AC4C7975B980'}
	(* Write text into an image. (expert function) *)
	FUNCTION F_VN_PutTextExp : HRESULT
	VAR_IN_OUT CONSTANT
		sText	:	STRING;	(* Text *)
	END_VAR
	VAR_INPUT
		ipDestImage	:	ITcVnImage;	(* Destination image *)
		nX	:	UDINT;	(* x coordinate (bottom left) *)
		nY	:	UDINT;	(* y coordinate (bottom left) *)
		eFontType	:	ETcVnFontType;	(* Font type *)
		fFontScale	:	LREAL;	(* Scaling factor *)
		aColor	:	REFERENCE TO TcVnVector4_LREAL;	(* Text color *)
		nThickness	:	DINT;	(* Line thickness *)
		eLineType	:	ETcVnLineType;	(* Line type *)
		bBottomLeftOrigin	:	BOOL;	(* Sets the image origin to the bottom left corner, if true *)
		hrPrev	:	HRESULT;	(* HRESULT indicating the result of previous operations (If SUCCEEDED(hrPrev) equals false, no operation is executed.) *)
	END_VAR

END_FUNCTION

// Functions/Keypoint Features/F_VN_FilterGoodMatches

	{attribute 'TcIecLibraryType'}
	{attribute 'external_name' := 'F_VN_FilterGoodMatches_GUID_EC15C148_9407_51B2_4E8A_F4A9388E2982'}
	(* Filter the descriptor matches and return only good ones. *)
	FUNCTION F_VN_FilterGoodMatches : HRESULT
	VAR_INPUT
		ipMatches	:	ITcVnContainer;	(* Container with descriptor matches (ContainerType_Vector_TcVnDMatch or ContainerType_Vector_Vector_TcVnDMatch) *)
		ipGoodMatches	:	REFERENCE TO ITcVnContainer;	(* Returns a container with good matches (ContainerType_Vector_TcVnDMatch) *)
		fMaxDist	:	REAL;	(* Maximum allowed descriptor distance (-1 disables this filter criterion) *)
		fMaxKnnRatio	:	REAL;	(* Maximum allowed distance ratio between first and second best match ([0..1], used for knn match results only, -1 disables this filter criterion) *)
		hrPrev	:	HRESULT;	(* HRESULT indicating the result of previous operations (If SUCCEEDED(hrPrev) equals false, no operation is executed.) *)
	END_VAR

END_FUNCTION

// Functions/Keypoint Features/F_VN_FindReferenceKeyPointsInImageORB

	{attribute 'TcIecLibraryType'}
	{attribute 'external_name' := 'F_VN_FindReferenceKeyPointsInImageORB_GUID_CBAD4079_436C_5DEE_5BB3_E82E6564762A'}
	(* Searches a reference image, represented by its ORB keypoints and corresponding descriptors, in a given source image (uses the default TcVnParamsORB parameters). *)
	FUNCTION F_VN_FindReferenceKeyPointsInImageORB : HRESULT
	VAR_INPUT
		ipSrcImage	:	ITcVnImage;	(* Source image *)
		ipRefKeyPoints	:	ITcVnContainer;	(* KeyPoints of the reference image, e.g. computed with F_VN_KeyPointsAndDescriptorsORB (ContainerType_Vector_TcVnKeyPoint) *)
		ipRefDescriptors	:	ITcVnImage;	(* Descriptors of the reference image KeyPoints, e.g. computed with F_VN_KeyPointsAndDescriptorsORB *)
		nRefImageWidth	:	UDINT;	(* Width of the reference image in pixels *)
		nRefImageHeight	:	UDINT;	(* Height of the reference image in pixels *)
		ipEdgePoints	:	REFERENCE TO ITcVnContainer;	(* Returns a container with the 4 edge points of the reference image transformed into ipSrcImage coordinates (ContainerType_Vector_TcVnPoint2_REAL) *)
		fMaxDist	:	REAL;	(* Maximum allowed descriptor distance (-1 disables this filter criterion) *)
		fMaxKnnRatio	:	REAL;	(* Maximum allowed distance ratio between first and second best match ([0..1], -1 disables this filter criterion) *)
		hrPrev	:	HRESULT;	(* HRESULT indicating the result of previous operations (If SUCCEEDED(hrPrev) equals false, no operation is executed.) *)
	END_VAR

END_FUNCTION

// Functions/Keypoint Features/F_VN_KeyPointsAndDescriptorsORB

	{attribute 'TcIecLibraryType'}
	{attribute 'external_name' := 'F_VN_KeyPointsAndDescriptorsORB_GUID_F30E1758_2201_586F_6DDD_1A40C364EA02'}
	(* Detects keypoints and compute descriptors using the ORB method. *)
	FUNCTION F_VN_KeyPointsAndDescriptorsORB : HRESULT
	VAR_INPUT
		ipSrcImage	:	ITcVnImage;	(* Source image *)
		ipKeyPoints	:	REFERENCE TO ITcVnContainer;	(* Returns a container which is filled with the keypoints (ContainerType_Vector_TcVnKeyPoint; Non-zero interface pointers are reused.) *)
		ipDescriptors	:	REFERENCE TO ITcVnImage;	(* Descriptor image (set to 0 if not required; 1 descriptor in each row; An appropriate image will be created if required.) *)
		hrPrev	:	HRESULT;	(* HRESULT indicating the result of previous operations (If SUCCEEDED(hrPrev) equals false, no operation is executed.) *)
	END_VAR

END_FUNCTION

// Functions/Keypoint Features/F_VN_FindReferenceKeyPointsInImageORBExp

	{attribute 'TcIecLibraryType'}
	{attribute 'external_name' := 'F_VN_FindReferenceKeyPointsInImageORBExp_GUID_16A9E510_1970_578F_5818_F43FD800F1CB'}
	(* Searches a reference image, represented by its ORB keypoints and corresponding descriptors, in a given source image. (expert function) *)
	FUNCTION F_VN_FindReferenceKeyPointsInImageORBExp : HRESULT
	VAR_INPUT
		ipSrcImage	:	ITcVnImage;	(* Source image *)
		ipRefKeyPoints	:	ITcVnContainer;	(* KeyPoints of the reference image, e.g. computed with F_VN_KeyPointsAndDescriptorsORB (ContainerType_Vector_TcVnKeyPoint) *)
		ipRefDescriptors	:	ITcVnImage;	(* Descriptors of the reference image KeyPoints, e.g. computed with F_VN_KeyPointsAndDescriptorsORB *)
		nRefImageWidth	:	UDINT;	(* Width of the reference image in pixels *)
		nRefImageHeight	:	UDINT;	(* Height of the reference image in pixels *)
		ipEdgePoints	:	REFERENCE TO ITcVnContainer;	(* Returns a container with the 4 edge points of the reference image transformed into ipSrcImage coordinates (ContainerType_Vector_TcVnPoint2_REAL) *)
		fMaxDist	:	REAL;	(* Maximum allowed descriptor distance (-1 disables this filter criterion) *)
		fMaxKnnRatio	:	REAL;	(* Maximum allowed distance ratio between first and second best match ([0..1], -1 disables this filter criterion) *)
		eNormType	:	ETcVnNormalizationType;	(* Normalization type used for descriptor matching (HAMMING recommended for ORB, HAMMING2 if the ORB nBriefPoints parameter is 3 or 4) *)
		ipSrcImageMask	:	ITcVnImage;	(* Mask to specify, where to look for keypoints in ipSrcImage (set to 0 if no mask required) *)
		stOrbParams	:	REFERENCE TO TcVnParamsORB;	(* Parameters to configure the keypoint and descriptor computation for ipSrcImage (resulting descriptors must be compatible to ipRefDescriptors!) *)
		eAlgorithm	:	ETcVnEstimationAlgorithm;	(* Estimation algorithm used for computing the perspective transformation between the two point sets *)
		fReprojThreshold	:	LREAL;	(* Maximum allowed reprojection error to treat a point pair as an inlier (only used if eAlgorithm is RANSAC, RHO) *)
		nMaxIterations	:	UDINT;	(* Maximum number of RANSAC iterations *)
		fConfidence	:	LREAL;	(* Confidence (0..1) *)
		hrPrev	:	HRESULT;	(* HRESULT indicating the result of previous operations (If SUCCEEDED(hrPrev) equals false, no operation is executed.) *)
	END_VAR

END_FUNCTION

// Functions/Keypoint Features/F_VN_KeyPointsAGAST

	{attribute 'TcIecLibraryType'}
	{attribute 'external_name' := 'F_VN_KeyPointsAGAST_GUID_E7453751_31AE_5C60_6CC1_514BF38E7BE8'}
	(* Detects keypoints using the AGAST method. *)
	FUNCTION F_VN_KeyPointsAGAST : HRESULT
	VAR_INPUT
		ipSrcImage	:	ITcVnImage;	(* Source image *)
		ipKeyPoints	:	REFERENCE TO ITcVnContainer;	(* Returns a container which is filled with the keypoints (ContainerType_Vector_TcVnKeyPoint; Non-zero interface pointers are reused.) *)
		hrPrev	:	HRESULT;	(* HRESULT indicating the result of previous operations (If SUCCEEDED(hrPrev) equals false, no operation is executed.) *)
	END_VAR

END_FUNCTION

// Functions/Keypoint Features/F_VN_KeyPointsAGASTExp

	{attribute 'TcIecLibraryType'}
	{attribute 'external_name' := 'F_VN_KeyPointsAGASTExp_GUID_F03F767C_BE67_5A4B_56FE_DCD207B4DF87'}
	(* Detects keypoints using the AGAST method. (expert function) *)
	FUNCTION F_VN_KeyPointsAGASTExp : HRESULT
	VAR_INPUT
		ipSrcImage	:	ITcVnImage;	(* Source image *)
		ipKeyPoints	:	REFERENCE TO ITcVnContainer;	(* Returns a container which is filled with the keypoints (ContainerType_Vector_TcVnKeyPoint; Non-zero interface pointers are reused.) *)
		ipMask	:	ITcVnImage;	(* Mask to specify, where to look for keypoints (set to 0 if no mask required) *)
		stParams	:	REFERENCE TO TcVnParamsAGAST;	(* Additional expert parameters *)
		hrPrev	:	HRESULT;	(* HRESULT indicating the result of previous operations (If SUCCEEDED(hrPrev) equals false, no operation is executed.) *)
	END_VAR

END_FUNCTION

// Functions/Keypoint Features/F_VN_KeyPointsAndDescriptorsAKAZE

	{attribute 'TcIecLibraryType'}
	{attribute 'external_name' := 'F_VN_KeyPointsAndDescriptorsAKAZE_GUID_5FA405E9_49FB_5F5A_5DDA_BB4EC4D0BADA'}
	(* Detects keypoints and compute descriptors using the AKAZE method. *)
	FUNCTION F_VN_KeyPointsAndDescriptorsAKAZE : HRESULT
	VAR_INPUT
		ipSrcImage	:	ITcVnImage;	(* Source image *)
		ipKeyPoints	:	REFERENCE TO ITcVnContainer;	(* Returns a container which is filled with the keypoints (ContainerType_Vector_TcVnKeyPoint; Non-zero interface pointers are reused.) *)
		ipDescriptors	:	REFERENCE TO ITcVnImage;	(* Descriptor image (set to 0 if not required; 1 descriptor in each row; An appropriate image will be created if required.) *)
		hrPrev	:	HRESULT;	(* HRESULT indicating the result of previous operations (If SUCCEEDED(hrPrev) equals false, no operation is executed.) *)
	END_VAR

END_FUNCTION

// Functions/Keypoint Features/F_VN_KeyPointsAndDescriptorsAKAZEExp

	{attribute 'TcIecLibraryType'}
	{attribute 'external_name' := 'F_VN_KeyPointsAndDescriptorsAKAZEExp_GUID_07AEC311_3D98_5509_615E_D1651924F5D6'}
	(* Detects keypoints and compute descriptors using the AKAZE method. (expert function) *)
	FUNCTION F_VN_KeyPointsAndDescriptorsAKAZEExp : HRESULT
	VAR_INPUT
		ipSrcImage	:	ITcVnImage;	(* Source image *)
		ipKeyPoints	:	REFERENCE TO ITcVnContainer;	(* Returns a container which is filled with the keypoints (ContainerType_Vector_TcVnKeyPoint; Non-zero interface pointers are reused.) *)
		ipDescriptors	:	REFERENCE TO ITcVnImage;	(* Descriptor image (set to 0 if not required; 1 descriptor in each row; An appropriate image will be created if required.) *)
		ipMask	:	ITcVnImage;	(* Mask to specify, where to look for keypoints (set to 0 if no mask required) *)
		stParams	:	REFERENCE TO TcVnParamsAKAZE;	(* Additional expert parameters *)
		hrPrev	:	HRESULT;	(* HRESULT indicating the result of previous operations (If SUCCEEDED(hrPrev) equals false, no operation is executed.) *)
	END_VAR

END_FUNCTION

// Functions/Keypoint Features/F_VN_KeyPointsAndDescriptorsBRISK

	{attribute 'TcIecLibraryType'}
	{attribute 'external_name' := 'F_VN_KeyPointsAndDescriptorsBRISK_GUID_E8984365_EC35_5908_6DCF_3812A28669DA'}
	(* Detects keypoints and compute descriptors using the BRISK method. *)
	FUNCTION F_VN_KeyPointsAndDescriptorsBRISK : HRESULT
	VAR_INPUT
		ipSrcImage	:	ITcVnImage;	(* Source image *)
		ipKeyPoints	:	REFERENCE TO ITcVnContainer;	(* Returns a container which is filled with the keypoints (ContainerType_Vector_TcVnKeyPoint; Non-zero interface pointers are reused.) *)
		ipDescriptors	:	REFERENCE TO ITcVnImage;	(* Descriptor image (set to 0 if not required; 1 descriptor in each row; An appropriate image will be created if required.) *)
		hrPrev	:	HRESULT;	(* HRESULT indicating the result of previous operations (If SUCCEEDED(hrPrev) equals false, no operation is executed.) *)
	END_VAR

END_FUNCTION

// Functions/Keypoint Features/F_VN_KeyPointsAndDescriptorsBRISKExp

	{attribute 'TcIecLibraryType'}
	{attribute 'external_name' := 'F_VN_KeyPointsAndDescriptorsBRISKExp_GUID_B63533A4_8E08_5EF5_43A0_D1C288E6355A'}
	(* Detects keypoints and compute descriptors using the BRISK method. (expert function) *)
	FUNCTION F_VN_KeyPointsAndDescriptorsBRISKExp : HRESULT
	VAR_INPUT
		ipSrcImage	:	ITcVnImage;	(* Source image *)
		ipKeyPoints	:	REFERENCE TO ITcVnContainer;	(* Returns a container which is filled with the keypoints (ContainerType_Vector_TcVnKeyPoint; Non-zero interface pointers are reused.) *)
		ipDescriptors	:	REFERENCE TO ITcVnImage;	(* Descriptor image (set to 0 if not required; 1 descriptor in each row; An appropriate image will be created if required.) *)
		ipMask	:	ITcVnImage;	(* Mask to specify, where to look for keypoints (set to 0 if no mask required) *)
		stParams	:	REFERENCE TO TcVnParamsBRISK;	(* Additional expert parameters *)
		hrPrev	:	HRESULT;	(* HRESULT indicating the result of previous operations (If SUCCEEDED(hrPrev) equals false, no operation is executed.) *)
	END_VAR

END_FUNCTION

// Functions/Keypoint Features/F_VN_KeyPointsAndDescriptorsKAZE

	{attribute 'TcIecLibraryType'}
	{attribute 'external_name' := 'F_VN_KeyPointsAndDescriptorsKAZE_GUID_A726C146_E174_53F0_5ED2_96C83DFCB1AA'}
	(* Detects keypoints and compute descriptors using the KAZE method. *)
	FUNCTION F_VN_KeyPointsAndDescriptorsKAZE : HRESULT
	VAR_INPUT
		ipSrcImage	:	ITcVnImage;	(* Source image *)
		ipKeyPoints	:	REFERENCE TO ITcVnContainer;	(* Returns a container which is filled with the keypoints (ContainerType_Vector_TcVnKeyPoint; Non-zero interface pointers are reused.) *)
		ipDescriptors	:	REFERENCE TO ITcVnImage;	(* Descriptor image (set to 0 if not required; 1 descriptor in each row; An appropriate image will be created if required.) *)
		hrPrev	:	HRESULT;	(* HRESULT indicating the result of previous operations (If SUCCEEDED(hrPrev) equals false, no operation is executed.) *)
	END_VAR

END_FUNCTION

// Functions/Keypoint Features/F_VN_KeyPointsAndDescriptorsKAZEExp

	{attribute 'TcIecLibraryType'}
	{attribute 'external_name' := 'F_VN_KeyPointsAndDescriptorsKAZEExp_GUID_C7959612_87EE_5F93_4D7C_D64A7BBFF46A'}
	(* Detects keypoints and compute descriptors using the KAZE method. (expert function) *)
	FUNCTION F_VN_KeyPointsAndDescriptorsKAZEExp : HRESULT
	VAR_INPUT
		ipSrcImage	:	ITcVnImage;	(* Source image *)
		ipKeyPoints	:	REFERENCE TO ITcVnContainer;	(* Returns a container which is filled with the keypoints (ContainerType_Vector_TcVnKeyPoint; Non-zero interface pointers are reused.) *)
		ipDescriptors	:	REFERENCE TO ITcVnImage;	(* Descriptor image (set to 0 if not required; 1 descriptor in each row; An appropriate image will be created if required.) *)
		ipMask	:	ITcVnImage;	(* Mask to specify, where to look for keypoints (set to 0 if no mask required) *)
		stParams	:	REFERENCE TO TcVnParamsKAZE;	(* Additional expert parameters *)
		hrPrev	:	HRESULT;	(* HRESULT indicating the result of previous operations (If SUCCEEDED(hrPrev) equals false, no operation is executed.) *)
	END_VAR

END_FUNCTION

// Functions/Keypoint Features/F_VN_KeyPointsAndDescriptorsORBExp

	{attribute 'TcIecLibraryType'}
	{attribute 'external_name' := 'F_VN_KeyPointsAndDescriptorsORBExp_GUID_8E96EEE0_57F1_507D_4CF8_B8895951513A'}
	(* Detect keypoints and compute descriptors using the ORB method. (expert function) *)
	FUNCTION F_VN_KeyPointsAndDescriptorsORBExp : HRESULT
	VAR_INPUT
		ipSrcImage	:	ITcVnImage;	(* Source image *)
		ipKeyPoints	:	REFERENCE TO ITcVnContainer;	(* Returns a container which is filled with the keypoints (ContainerType_Vector_TcVnKeyPoint; Non-zero interface pointers are reused.) *)
		ipDescriptors	:	REFERENCE TO ITcVnImage;	(* Descriptor image (set to 0 if not required; 1 descriptor in each row; An appropriate image will be created if required.) *)
		ipMask	:	ITcVnImage;	(* Mask to specify, where to look for keypoints (set to 0 if no mask required) *)
		stParams	:	REFERENCE TO TcVnParamsORB;	(* Additional expert parameters *)
		hrPrev	:	HRESULT;	(* HRESULT indicating the result of previous operations (If SUCCEEDED(hrPrev) equals false, no operation is executed.) *)
	END_VAR

END_FUNCTION

// Functions/Keypoint Features/F_VN_KeyPointsFAST

	{attribute 'TcIecLibraryType'}
	{attribute 'external_name' := 'F_VN_KeyPointsFAST_GUID_3F9E7E53_CA5F_50E7_6478_729EF955EBF6'}
	(* Detects keypoints using the FAST method. *)
	FUNCTION F_VN_KeyPointsFAST : HRESULT
	VAR_INPUT
		ipSrcImage	:	ITcVnImage;	(* Source image (single-channel). *)
		ipKeyPoints	:	REFERENCE TO ITcVnContainer;	(* Returns a container which is filled with the keypoints (ContainerType_Vector_TcVnKeyPoint; Non-zero interface pointers are reused.) *)
		hrPrev	:	HRESULT;	(* HRESULT indicating the result of previous operations (If SUCCEEDED(hrPrev) equals false, no operation is executed.) *)
	END_VAR

END_FUNCTION

// Functions/Keypoint Features/F_VN_KeyPointsFASTExp

	{attribute 'TcIecLibraryType'}
	{attribute 'external_name' := 'F_VN_KeyPointsFASTExp_GUID_E544DD38_DC15_5753_7BB4_1E6EAE2BCA03'}
	(* Detects keypoints using the FAST method. (expert function) *)
	FUNCTION F_VN_KeyPointsFASTExp : HRESULT
	VAR_INPUT
		ipSrcImage	:	ITcVnImage;	(* Source image *)
		ipKeyPoints	:	REFERENCE TO ITcVnContainer;	(* Returns a container which is filled with the keypoints (ContainerType_Vector_TcVnKeyPoint; Non-zero interface pointers are reused.) *)
		ipMask	:	ITcVnImage;	(* Mask to specify, where to look for keypoints (set to 0 if no mask required) *)
		stParams	:	REFERENCE TO TcVnParamsFAST;	(* Additional expert parameters *)
		hrPrev	:	HRESULT;	(* HRESULT indicating the result of previous operations (If SUCCEEDED(hrPrev) equals false, no operation is executed.) *)
	END_VAR

END_FUNCTION

// Functions/Keypoint Features/F_VN_KeyPointsGFTT

	{attribute 'TcIecLibraryType'}
	{attribute 'external_name' := 'F_VN_KeyPointsGFTT_GUID_271B9ACD_5DD6_5584_5AE8_66922A81BD72'}
	(* Detects keypoints using the GFTT method, which detects strong corners. *)
	FUNCTION F_VN_KeyPointsGFTT : HRESULT
	VAR_INPUT
		ipSrcImage	:	ITcVnImage;	(* Source image *)
		ipKeyPoints	:	REFERENCE TO ITcVnContainer;	(* Returns a container which is filled with the keypoints (ContainerType_Vector_TcVnKeyPoint; Non-zero interface pointers are reused.) *)
		hrPrev	:	HRESULT;	(* HRESULT indicating the result of previous operations (If SUCCEEDED(hrPrev) equals false, no operation is executed.) *)
	END_VAR

END_FUNCTION

// Functions/Keypoint Features/F_VN_KeyPointsGFTTExp

